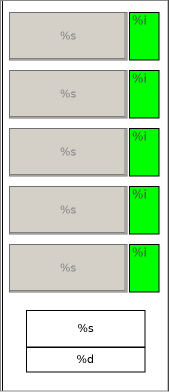
VISUALIZATION VISU_AXE_STD1_FCT_OP  // 169x392
VAR_IN_OUT
	m_Input_MOTEUR: BLOCK_AXE_STD1;
	m_Input_PRG_MOUVEMENT_PS: BLOCK_PRG_MOUVEMENT_PS;
END_VAR
VAR_INPUT
	m_Input_INDEX_MOTEUR : INT;
END_VAR
    RoundedRectangle (2,-1 167x392)
    Rectangle (26,310 119x37), "%s", invisible if: NOT m_Input_PRG_MOUVEMENT_PS.CONF_Balayage[m_Input_INDEX_MOTEUR], text list: 'TextList_Moteurs', text index: 3
    Rectangle (26,347 119x25), "%d", text variable: m_Input_MOTEUR.STATE_NBal, invisible if: NOT m_Input_PRG_MOUVEMENT_PS.CONF_Balayage[m_Input_INDEX_MOTEUR]
    Frame (9,12 152x50)
        shows VISU_FCTS_SA(m_Input_ID_XML := 6, m_Input_Operation := m_Input_MOTEUR.OP_Validation, m_Input_UserRight := PRG_USER.ACTU_USER.FONCTION_SA)
    Frame (9,70 152x50)
        shows VISU_FCTS_SA(m_Input_ID_XML := 7, m_Input_Operation := m_Input_MOTEUR.OP_Stop, m_Input_UserRight := PRG_USER.ACTU_USER.FONCTION_SA)
    Frame (9,128 152x50), invisible if: NOT m_Input_PRG_MOUVEMENT_PS.CONF_Positionnement[m_Input_INDEX_MOTEUR]
        shows VISU_FCTS_SA(m_Input_ID_XML := 8, m_Input_Operation := m_Input_MOTEUR.OP_Position, m_Input_UserRight := PRG_USER.ACTU_USER.FONCTION_SA)
    Frame (9,186 152x50), invisible if: NOT m_Input_PRG_MOUVEMENT_PS.CONF_Rotation[m_Input_INDEX_MOTEUR]
        shows VISU_FCTS_SA(m_Input_ID_XML := 15, m_Input_Operation := m_Input_MOTEUR.OP_Rotation, m_Input_UserRight := PRG_USER.ACTU_USER.FONCTION_SA)
    Frame (9,244 152x50), invisible if: NOT m_Input_PRG_MOUVEMENT_PS.CONF_Balayage[m_Input_INDEX_MOTEUR]
        shows VISU_FCTS_SA(m_Input_ID_XML := 16, m_Input_Operation := m_Input_MOTEUR.OP_Balayage, m_Input_UserRight := PRG_USER.ACTU_USER.FONCTION_SA)
END_VISUALIZATION

// ---- Visualizations/Symbole/MOUVEMENTS PS/AXE STD1/FCT_Part/VISU_AXE_STD1_FCT_OP_OSC.TcVIS
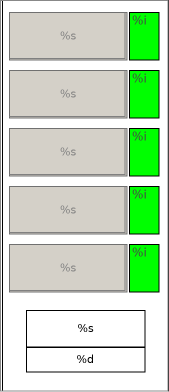
VISUALIZATION VISU_AXE_STD1_FCT_OP_OSC  // 169x392
VAR_IN_OUT
	m_Input_MOTEUR: BLOCK_AXE_STD1_OSCILLANT;
	m_Input_PRG_MOUVEMENT_PS: BLOCK_PRG_MOUVEMENT_PS;
END_VAR
VAR_INPUT
	m_Input_INDEX_MOTEUR : INT;
END_VAR
    RoundedRectangle (2,-1 167x392)
    Rectangle (26,310 119x37), "%s", invisible if: NOT m_Input_PRG_MOUVEMENT_PS.CONF_Balayage[m_Input_INDEX_MOTEUR], text list: 'TextList_Moteurs', text index: 3
    Rectangle (26,347 119x25), "%d", text variable: m_Input_MOTEUR.STATE_NBal, invisible if: NOT m_Input_PRG_MOUVEMENT_PS.CONF_Balayage[m_Input_INDEX_MOTEUR]
    Frame (9,12 152x50)
        shows VISU_FCTS_SA(m_Input_ID_XML := 6, m_Input_Operation := m_Input_MOTEUR.OP_Validation, m_Input_UserRight := PRG_USER.ACTU_USER.FONCTION_SA)
    Frame (9,70 152x50)
        shows VISU_FCTS_SA(m_Input_ID_XML := 7, m_Input_Operation := m_Input_MOTEUR.OP_Stop, m_Input_UserRight := PRG_USER.ACTU_USER.FONCTION_SA)
    Frame (9,128 152x50), invisible if: NOT m_Input_PRG_MOUVEMENT_PS.CONF_Positionnement[m_Input_INDEX_MOTEUR]
        shows VISU_FCTS_SA(m_Input_ID_XML := 8, m_Input_Operation := m_Input_MOTEUR.OP_Position, m_Input_UserRight := PRG_USER.ACTU_USER.FONCTION_SA)
    Frame (9,186 152x50), invisible if: NOT m_Input_PRG_MOUVEMENT_PS.CONF_Rotation[m_Input_INDEX_MOTEUR]
        shows VISU_FCTS_SA(m_Input_ID_XML := 15, m_Input_Operation := m_Input_MOTEUR.OP_Rotation, m_Input_UserRight := PRG_USER.ACTU_USER.FONCTION_SA)
    Frame (9,244 152x50), invisible if: NOT m_Input_PRG_MOUVEMENT_PS.CONF_Balayage[m_Input_INDEX_MOTEUR]
        shows VISU_FCTS_SA(m_Input_ID_XML := 16, m_Input_Operation := m_Input_MOTEUR.OP_Balayage, m_Input_UserRight := PRG_USER.ACTU_USER.FONCTION_SA)
END_VISUALIZATION

// ---- Visualizations/Symbole/MOUVEMENTS PS/AXE STD1/FCT_Part/VISU_AXE_STD1_FCT_TRF.TcVIS
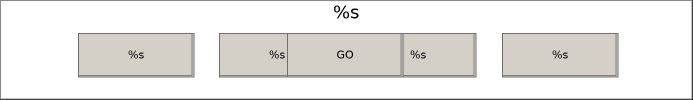
VISUALIZATION VISU_AXE_STD1_FCT_TRF  // 693x100
VAR_IN_OUT
	m_Input_MOTEUR: BLOCK_AXE_STD1;
	m_Input_PRG_MOUVEMENT_PS: BLOCK_PRG_MOUVEMENT_PS;
END_VAR
VAR_INPUT CONSTANT
	m_Input_INDEX_MOTEUR : INT;
	m_Input_Ref_Trf:		USINT;
END_VAR
    Rectangle (0,0 693x100), "%s", text list: 'TextList_Moteurs', text index: 4
    Button (78,33 116x44), "%s", text variable: m_Input_MOTEUR.CONF_ID_Poste[1], invisible if: m_Input_PRG_MOUVEMENT_PS.CONF_NB_POSTE[m_Input_INDEX_MOTEUR]<1, input disabled if: NOT m_Input_MOTEUR.OP_Position.AUTOR_IHM
        OnMouseClick: execute {
            m_Input_MOTEUR.PRM_NPOSTE:=1;
            m_Input_MOTEUR.PRM_NREF:=m_Input_REF_TRF;
            m_Input_MOTEUR.PRM_BalPos:=FALSE;
            m_Input_MOTEUR.PRM_GoToHome:=TRUE;
            m_Input_MOTEUR.PRM_Position:=0;
            m_Input_MOTEUR.OP_POSITION.ON_IHM:=TRUE;
        }
    Button (219,33 116x44), "%s", text variable: m_Input_MOTEUR.CONF_ID_Poste[2], invisible if: m_Input_PRG_MOUVEMENT_PS.CONF_NB_POSTE[m_Input_INDEX_MOTEUR]<2, input disabled if: NOT m_Input_MOTEUR.OP_Position.AUTOR_IHM
        OnMouseClick: execute {
            m_Input_MOTEUR.PRM_NPOSTE:=2;
            m_Input_MOTEUR.PRM_NREF:=m_Input_REF_TRF;
            m_Input_MOTEUR.PRM_BalPos:=FALSE;
            m_Input_MOTEUR.PRM_GoToHome:=TRUE;
            m_Input_MOTEUR.PRM_Position:=0;
            m_Input_MOTEUR.OP_POSITION.ON_IHM:=TRUE;
        }
    Button (360,33 116x44), "%s", text variable: m_Input_MOTEUR.CONF_ID_Poste[3], invisible if: m_Input_PRG_MOUVEMENT_PS.CONF_NB_POSTE[m_Input_INDEX_MOTEUR]<3, input disabled if: NOT m_Input_MOTEUR.OP_Position.AUTOR_IHM
        OnMouseClick: execute {
            m_Input_MOTEUR.PRM_NPOSTE:=3;
            m_Input_MOTEUR.PRM_NREF:=m_Input_REF_TRF;
            m_Input_MOTEUR.PRM_BalPos:=FALSE;
            m_Input_MOTEUR.PRM_GoToHome:=TRUE;
            m_Input_MOTEUR.PRM_Position:=0;
            m_Input_MOTEUR.OP_POSITION.ON_IHM:=TRUE;
        }
    Button (502,33 116x44), "%s", text variable: m_Input_MOTEUR.CONF_ID_Poste[4], invisible if: m_Input_PRG_MOUVEMENT_PS.CONF_NB_POSTE[m_Input_INDEX_MOTEUR]<4, input disabled if: NOT m_Input_MOTEUR.OP_Position.AUTOR_IHM
        OnMouseClick: execute {
            m_Input_MOTEUR.PRM_NPOSTE:=4;
            m_Input_MOTEUR.PRM_NREF:=m_Input_REF_TRF;
            m_Input_MOTEUR.PRM_BalPos:=FALSE;
            m_Input_MOTEUR.PRM_GoToHome:=TRUE;
            m_Input_MOTEUR.PRM_Position:=0;
            m_Input_MOTEUR.OP_POSITION.ON_IHM:=TRUE;
        }
    Button (287,33 116x44), "GO", invisible if: m_Input_PRG_MOUVEMENT_PS.CONF_NB_POSTE[m_Input_INDEX_MOTEUR]<>0, input disabled if: NOT m_Input_MOTEUR.OP_Position.AUTOR_IHM
        OnMouseClick: execute {
            m_Input_MOTEUR.PRM_NPOSTE:=0;
            m_Input_MOTEUR.PRM_NREF:=0;
            m_Input_MOTEUR.PRM_BalPos:=FALSE;
            m_Input_MOTEUR.PRM_GoToHome:=TRUE;
            m_Input_MOTEUR.PRM_Position:=0;
            m_Input_MOTEUR.OP_POSITION.ON_IHM:=TRUE;
        }
END_VISUALIZATION

// ---- Visualizations/Symbole/MOUVEMENTS PS/AXE STD1/FCT_Part/VISU_AXE_STD1_FCT_TRF_OSC.TcVIS
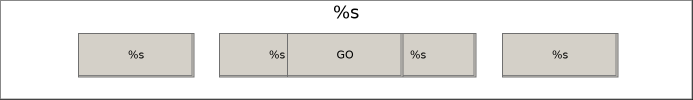
VISUALIZATION VISU_AXE_STD1_FCT_TRF_OSC  // 693x100
VAR_IN_OUT
	m_Input_MOTEUR: BLOCK_AXE_STD1_OSCILLANT;
	m_Input_PRG_MOUVEMENT_PS: BLOCK_PRG_MOUVEMENT_PS;
END_VAR
VAR_INPUT CONSTANT
	m_Input_INDEX_MOTEUR : INT;
	m_Input_Ref_Trf:		USINT;
END_VAR
    Rectangle (0,0 693x100), "%s", text list: 'TextList_Moteurs', text index: 4
    Button (78,33 116x44), "%s", text variable: m_Input_MOTEUR.CONF_ID_Poste[1], invisible if: m_Input_PRG_MOUVEMENT_PS.CONF_NB_POSTE[m_Input_INDEX_MOTEUR]<1, input disabled if: NOT m_Input_MOTEUR.OP_Position.AUTOR_IHM
        OnMouseClick: execute {
            m_Input_MOTEUR.PRM_NPOSTE:=1;
            m_Input_MOTEUR.PRM_NREF:=m_Input_REF_TRF;
            m_Input_MOTEUR.PRM_BalPos:=FALSE;
            m_Input_MOTEUR.PRM_GoToHome:=TRUE;
            m_Input_MOTEUR.PRM_Position:=0;
            m_Input_MOTEUR.OP_POSITION.ON_IHM:=TRUE;
        }
    Button (219,33 116x44), "%s", text variable: m_Input_MOTEUR.CONF_ID_Poste[2], invisible if: m_Input_PRG_MOUVEMENT_PS.CONF_NB_POSTE[m_Input_INDEX_MOTEUR]<2, input disabled if: NOT m_Input_MOTEUR.OP_Position.AUTOR_IHM
        OnMouseClick: execute {
            m_Input_MOTEUR.PRM_NPOSTE:=2;
            m_Input_MOTEUR.PRM_NREF:=m_Input_REF_TRF;
            m_Input_MOTEUR.PRM_BalPos:=FALSE;
            m_Input_MOTEUR.PRM_GoToHome:=TRUE;
            m_Input_MOTEUR.PRM_Position:=0;
            m_Input_MOTEUR.OP_POSITION.ON_IHM:=TRUE;
        }
    Button (360,33 116x44), "%s", text variable: m_Input_MOTEUR.CONF_ID_Poste[3], invisible if: m_Input_PRG_MOUVEMENT_PS.CONF_NB_POSTE[m_Input_INDEX_MOTEUR]<3, input disabled if: NOT m_Input_MOTEUR.OP_Position.AUTOR_IHM
        OnMouseClick: execute {
            m_Input_MOTEUR.PRM_NPOSTE:=3;
            m_Input_MOTEUR.PRM_NREF:=m_Input_REF_TRF;
            m_Input_MOTEUR.PRM_BalPos:=FALSE;
            m_Input_MOTEUR.PRM_GoToHome:=TRUE;
            m_Input_MOTEUR.PRM_Position:=0;
            m_Input_MOTEUR.OP_POSITION.ON_IHM:=TRUE;
        }
    Button (502,33 116x44), "%s", text variable: m_Input_MOTEUR.CONF_ID_Poste[4], invisible if: m_Input_PRG_MOUVEMENT_PS.CONF_NB_POSTE[m_Input_INDEX_MOTEUR]<4, input disabled if: NOT m_Input_MOTEUR.OP_Position.AUTOR_IHM
        OnMouseClick: execute {
            m_Input_MOTEUR.PRM_NPOSTE:=4;
            m_Input_MOTEUR.PRM_NREF:=m_Input_REF_TRF;
            m_Input_MOTEUR.PRM_BalPos:=FALSE;
            m_Input_MOTEUR.PRM_GoToHome:=TRUE;
            m_Input_MOTEUR.PRM_Position:=0;
            m_Input_MOTEUR.OP_POSITION.ON_IHM:=TRUE;
        }
    Button (287,33 116x44), "GO", invisible if: m_Input_PRG_MOUVEMENT_PS.CONF_NB_POSTE[m_Input_INDEX_MOTEUR]<>0, input disabled if: NOT m_Input_MOTEUR.OP_Position.AUTOR_IHM
        OnMouseClick: execute {
            m_Input_MOTEUR.PRM_NPOSTE:=0;
            m_Input_MOTEUR.PRM_NREF:=0;
            m_Input_MOTEUR.PRM_BalPos:=FALSE;
            m_Input_MOTEUR.PRM_GoToHome:=TRUE;
            m_Input_MOTEUR.PRM_Position:=0.0;
            m_Input_MOTEUR.OP_POSITION.ON_IHM:=TRUE;
        }
END_VISUALIZATION

// ---- Visualizations/Symbole/MOUVEMENTS PS/AXE STD1/FCT_Part/VISU_AXE_STD1_LIN_REL_FCT_ETAT.TcVIS
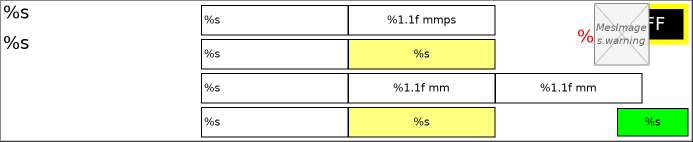
VISUALIZATION VISU_AXE_STD1_LIN_REL_FCT_ETAT  // 693x142
VAR_IN_OUT
	m_Input_MOTEUR: BLOCK_AXE_STD1;
	m_Input_PRG_MOUVEMENT_PS: BLOCK_PRG_MOUVEMENT_PS;
END_VAR
VAR_INPUT
	m_Input_ID_NOM_XML : INT;
END_VAR
    Rectangle (0,0 693x142), "%s", text list: 'TextList_Type_Moteur', text index: m_Input_ID_NOM_XML
    Rectangle (0,28 107x30), "%s", text variable: m_Input_MOTEUR.MNEMO
    RoundedRectangle (201,5 147x30), "%s", text list: 'TextList_Moteurs', text index: 7
    RoundedRectangle (201,39 147x30), "%s", text list: 'TextList_Moteurs', text index: 8
    RoundedRectangle (201,73 147x30), "%s", text list: 'TextList_Moteurs', text index: 9
    RoundedRectangle (201,107 147x30), "%s", text list: 'TextList_Moteurs', text index: 10
    RoundedRectangle (348,5 147x30), "%1.1f mmps", text variable: m_Input_MOTEUR.STATE_Vit
    RoundedRectangle (348,39 147x30), "%s", text variable: m_Input_MOTEUR.CONF_ID_POSTE[m_Input_MOTEUR.PRM_NPOSTE]
    RoundedRectangle (348,73 147x30), "%1.1f mm", text variable: m_Input_MOTEUR.STATE_Pos_Rel
    RoundedRectangle (495,73 147x30), "%1.1f mm", text variable: m_Input_MOTEUR.STATE_Pos
    RoundedRectangle (348,107 147x30), "%s", text variable: m_Input_MOTEUR.CONF_ID_REF[m_Input_MOTEUR.PRM_NRef]
    RoundedRectangle (617,108 71x28), "%s", invisible if: m_Input_MOTEUR.STATE_Homed OR m_Input_MOTEUR.CONF_No_Ref, text list: 'TextList_Moteurs', text index: 11
    RoundedRectangle (617,108 71x28), "%s", invisible if: NOT m_Input_MOTEUR.STATE_Homed OR m_Input_MOTEUR.CONF_No_Ref, text list: 'TextList_Moteurs', text index: 11
    RoundedRectangle (608,4 80x40), invisible if: NOT m_Input_MOTEUR.OP_Validation.OK
    RoundedRectangle (608,4 80x40), invisible if: NOT m_Input_MOTEUR.OP_Validation.AR
    RoundedRectangle (608,4 80x40), invisible if: NOT m_Input_MOTEUR.OP_Validation.EC
    RoundedRectangle (613,9 70x30), "ON", invisible if: m_Input_MOTEUR.STATE_Ar
    RoundedRectangle (613,9 70x30), "OFF", invisible if: NOT m_Input_MOTEUR.STATE_Ar
    Rectangle (535,24 67x21), "%i", text variable: m_Input_MOTEUR.STATE_Err, invisible if: NOT m_Input_MOTEUR.STATE_NOK
    Image (594,3 55x62), invisible if: NOT m_Input_MOTEUR.STATE_NOK, image: MesImages.warning
END_VISUALIZATION

// ---- Visualizations/Symbole/MOUVEMENTS PS/AXE STD1/FCT_Part/VISU_AXE_STD1_LIN_REL_FCT_ETAT_OSC.TcVIS
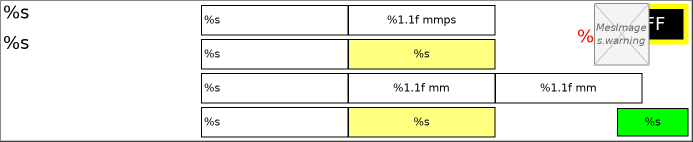
VISUALIZATION VISU_AXE_STD1_LIN_REL_FCT_ETAT_OSC  // 693x142
VAR_IN_OUT
	m_Input_MOTEUR: BLOCK_AXE_STD1_OSCILLANT;
	m_Input_PRG_MOUVEMENT_PS: BLOCK_PRG_MOUVEMENT_PS;
END_VAR
VAR_INPUT
	m_Input_ID_NOM_XML : INT;
END_VAR
    Rectangle (0,0 693x142), "%s", text list: 'TextList_Type_Moteur', text index: m_Input_ID_NOM_XML
    Rectangle (0,28 107x30), "%s", text variable: m_Input_MOTEUR.MNEMO
    RoundedRectangle (201,5 147x30), "%s", text list: 'TextList_Moteurs', text index: 7
    RoundedRectangle (201,39 147x30), "%s", text list: 'TextList_Moteurs', text index: 8
    RoundedRectangle (201,73 147x30), "%s", text list: 'TextList_Moteurs', text index: 9
    RoundedRectangle (201,107 147x30), "%s", text list: 'TextList_Moteurs', text index: 10
    RoundedRectangle (348,5 147x30), "%1.1f mmps", text variable: m_Input_MOTEUR.STATE_Vit
    RoundedRectangle (348,39 147x30), "%s", text variable: m_Input_MOTEUR.CONF_ID_POSTE[m_Input_MOTEUR.PRM_NPOSTE]
    RoundedRectangle (348,73 147x30), "%1.1f mm", text variable: m_Input_MOTEUR.STATE_Pos_Rel
    RoundedRectangle (495,73 147x30), "%1.1f mm", text variable: m_Input_MOTEUR.STATE_Pos
    RoundedRectangle (348,107 147x30), "%s", text variable: m_Input_MOTEUR.CONF_ID_REF[m_Input_MOTEUR.PRM_NRef]
    RoundedRectangle (617,108 71x28), "%s", invisible if: m_Input_MOTEUR.STATE_Homed OR m_Input_MOTEUR.CONF_No_Ref, text list: 'TextList_Moteurs', text index: 11
    RoundedRectangle (617,108 71x28), "%s", invisible if: NOT m_Input_MOTEUR.STATE_Homed OR m_Input_MOTEUR.CONF_No_Ref, text list: 'TextList_Moteurs', text index: 11
    RoundedRectangle (608,4 80x40), invisible if: NOT m_Input_MOTEUR.OP_Validation.OK
    RoundedRectangle (608,4 80x40), invisible if: NOT m_Input_MOTEUR.OP_Validation.AR
    RoundedRectangle (608,4 80x40), invisible if: NOT m_Input_MOTEUR.OP_Validation.EC
    RoundedRectangle (613,9 70x30), "ON", invisible if: m_Input_MOTEUR.STATE_Ar
    RoundedRectangle (613,9 70x30), "OFF", invisible if: NOT m_Input_MOTEUR.STATE_Ar
    Rectangle (535,24 67x21), "%i", text variable: m_Input_MOTEUR.STATE_Err, invisible if: NOT m_Input_MOTEUR.STATE_NOK
    Image (594,3 55x62), invisible if: NOT m_Input_MOTEUR.STATE_NOK, image: MesImages.warning
END_VISUALIZATION

// ---- Visualizations/Symbole/MOUVEMENTS PS/AXE STD1/FCT_Part/VISU_AXE_STD1_LIN_ROT_FCT_CONS.TcVIS
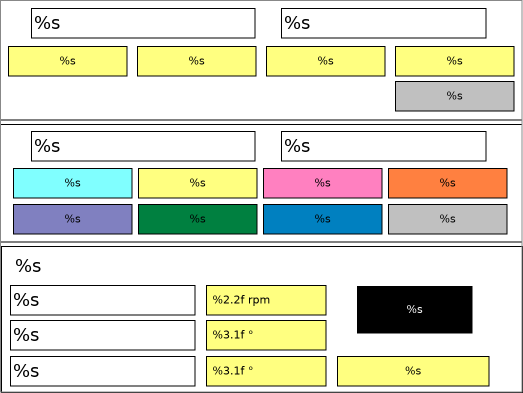
VISUALIZATION VISU_AXE_STD1_LIN_ROT_FCT_CONS  // 523x393
VAR_IN_OUT
	m_Input_MOTEUR: BLOCK_AXE_STD1;
	m_Input_PRG_MOUVEMENT_PS: BLOCK_PRG_MOUVEMENT_PS;
END_VAR
VAR_INPUT CONSTANT
	m_Input_INDEX_MOTEUR : INT;
END_VAR
    Rectangle (0,0 522x120)
    RoundedRectangle (31,8 224x30), "%s", text list: 'TextList_Moteurs', text index: 13
    RoundedRectangle (281,8 205x30), "%s", text variable: m_Input_MOTEUR.CONF_ID_Poste[m_Input_MOTEUR.PRM_NPoste]
    RoundedRectangle (8,46 119x30), "%s", text variable: m_Input_MOTEUR.CONF_ID_Poste[1], invisible if: m_Input_PRG_MOUVEMENT_PS.CONF_NB_POSTE[m_Input_INDEX_MOTEUR]<1, input disabled if: (NOT PRG_User.ACTU_USER.MAINTENANCE AND m_Input_MOTEUR.MANUAL) OR (NOT PRG_User.ACTU_USER.FONCTION_SA AND NOT m_Input_MOTEUR.MANUAL)
        OnMouseClick: execute { m_Input_MOTEUR.PRM_NPOSTE:=1; }
    RoundedRectangle (395,81 119x30), "%s", text variable: m_Input_MOTEUR.CONF_ID_POSTE[0], invisible if: NOT m_Input_PRG_MOUVEMENT_PS.CONF_Use_Poste0[m_Input_INDEX_MOTEUR], input disabled if: (NOT PRG_User.ACTU_USER.MAINTENANCE AND m_Input_MOTEUR.MANUAL) OR (NOT PRG_User.ACTU_USER.FONCTION_SA AND NOT m_Input_MOTEUR.MANUAL)
        OnMouseClick: execute { m_Input_MOTEUR.PRM_NPOSTE:=0; }
    RoundedRectangle (137,46 119x30), "%s", text variable: m_Input_MOTEUR.CONF_ID_Poste[2], invisible if: m_Input_PRG_MOUVEMENT_PS.CONF_NB_POSTE[m_Input_INDEX_MOTEUR]<2, input disabled if: (NOT PRG_User.ACTU_USER.MAINTENANCE AND m_Input_MOTEUR.MANUAL) OR (NOT PRG_User.ACTU_USER.FONCTION_SA AND NOT m_Input_MOTEUR.MANUAL)
        OnMouseClick: execute { m_Input_MOTEUR.PRM_NPOSTE:=2; }
    RoundedRectangle (266,46 119x30), "%s", text variable: m_Input_MOTEUR.CONF_ID_Poste[3], invisible if: m_Input_PRG_MOUVEMENT_PS.CONF_NB_POSTE[m_Input_INDEX_MOTEUR]<3, input disabled if: (NOT PRG_User.ACTU_USER.MAINTENANCE AND m_Input_MOTEUR.MANUAL) OR (NOT PRG_User.ACTU_USER.FONCTION_SA AND NOT m_Input_MOTEUR.MANUAL)
        OnMouseClick: execute { m_Input_MOTEUR.PRM_NPOSTE:=3; }
    RoundedRectangle (395,46 119x30), "%s", text variable: m_Input_MOTEUR.CONF_ID_Poste[4], invisible if: m_Input_PRG_MOUVEMENT_PS.CONF_NB_POSTE[m_Input_INDEX_MOTEUR]<4, input disabled if: (NOT PRG_User.ACTU_USER.MAINTENANCE AND m_Input_MOTEUR.MANUAL) OR (NOT PRG_User.ACTU_USER.FONCTION_SA AND NOT m_Input_MOTEUR.MANUAL)
        OnMouseClick: execute { m_Input_MOTEUR.PRM_NPOSTE:=4; }
    Rectangle (0,124 522x118)
    RoundedRectangle (31,131 224x30), "%s", text list: 'TextList_Moteurs', text index: 14
    RoundedRectangle (281,131 205x30), "%s", text variable: m_Input_MOTEUR.CONF_ID_Ref[m_Input_MOTEUR.PRM_NRef]
    RoundedRectangle (13,168 119x30), "%s", text variable: m_Input_MOTEUR.CONF_ID_REF[1], invisible if: m_Input_PRG_MOUVEMENT_PS.CONF_NB_REF[m_Input_INDEX_MOTEUR]<1, input disabled if: (NOT PRG_User.ACTU_USER.MAINTENANCE AND m_Input_MOTEUR.MANUAL) OR (NOT PRG_User.ACTU_USER.FONCTION_SA AND NOT m_Input_MOTEUR.MANUAL)
        OnMouseClick: execute { m_Input_MOTEUR.PRM_NREF:=1; }
    RoundedRectangle (138,168 119x30), "%s", text variable: m_Input_MOTEUR.CONF_ID_REF[2], invisible if: m_Input_PRG_MOUVEMENT_PS.CONF_NB_REF[m_Input_INDEX_MOTEUR]<2, input disabled if: (NOT PRG_User.ACTU_USER.MAINTENANCE AND m_Input_MOTEUR.MANUAL) OR (NOT PRG_User.ACTU_USER.FONCTION_SA AND NOT m_Input_MOTEUR.MANUAL)
        OnMouseClick: execute { m_Input_MOTEUR.PRM_NREF:=2; }
    RoundedRectangle (263,168 119x30), "%s", text variable: m_Input_MOTEUR.CONF_ID_REF[3], invisible if: m_Input_PRG_MOUVEMENT_PS.CONF_NB_REF[m_Input_INDEX_MOTEUR]<3, input disabled if: (NOT PRG_User.ACTU_USER.MAINTENANCE AND m_Input_MOTEUR.MANUAL) OR (NOT PRG_User.ACTU_USER.FONCTION_SA AND NOT m_Input_MOTEUR.MANUAL)
        OnMouseUp: execute { m_Input_MOTEUR.PRM_NREF:=3; }
    RoundedRectangle (388,168 119x30), "%s", text variable: m_Input_MOTEUR.CONF_ID_REF[4], invisible if: m_Input_PRG_MOUVEMENT_PS.CONF_NB_REF[m_Input_INDEX_MOTEUR]<4, input disabled if: (NOT PRG_User.ACTU_USER.MAINTENANCE AND m_Input_MOTEUR.MANUAL) OR (NOT PRG_User.ACTU_USER.FONCTION_SA AND NOT m_Input_MOTEUR.MANUAL)
        OnMouseClick: execute { m_Input_MOTEUR.PRM_NREF:=4; }
    RoundedRectangle (13,204 119x30), "%s", text variable: m_Input_MOTEUR.CONF_ID_REF[5], invisible if: m_Input_PRG_MOUVEMENT_PS.CONF_NB_REF[m_Input_INDEX_MOTEUR]<5, input disabled if: (NOT PRG_User.ACTU_USER.MAINTENANCE AND m_Input_MOTEUR.MANUAL) OR (NOT PRG_User.ACTU_USER.FONCTION_SA AND NOT m_Input_MOTEUR.MANUAL)
        OnMouseClick: execute { m_Input_MOTEUR.PRM_NREF:=5; }
    RoundedRectangle (138,204 119x30), "%s", text variable: m_Input_MOTEUR.CONF_ID_REF[6], invisible if: m_Input_PRG_MOUVEMENT_PS.CONF_NB_REF[m_Input_INDEX_MOTEUR]<6, input disabled if: (NOT PRG_User.ACTU_USER.MAINTENANCE AND m_Input_MOTEUR.MANUAL) OR (NOT PRG_User.ACTU_USER.FONCTION_SA AND NOT m_Input_MOTEUR.MANUAL)
        OnMouseClick: execute { m_Input_MOTEUR.PRM_NREF:=6; }
    RoundedRectangle (388,204 119x30), "%s", text variable: m_Input_MOTEUR.CONF_ID_REF[0], invisible if: NOT m_Input_PRG_MOUVEMENT_PS.CONF_Use_Ref0[m_Input_INDEX_MOTEUR], input disabled if: (NOT PRG_User.ACTU_USER.MAINTENANCE AND m_Input_MOTEUR.MANUAL) OR (NOT PRG_User.ACTU_USER.FONCTION_SA AND NOT m_Input_MOTEUR.MANUAL)
        OnMouseClick: execute { m_Input_MOTEUR.PRM_NREF:=0; }
    RoundedRectangle (263,204 119x30), "%s", text variable: m_Input_MOTEUR.CONF_ID_REF[7], invisible if: m_Input_PRG_MOUVEMENT_PS.CONF_NB_REF[m_Input_INDEX_MOTEUR]<7, input disabled if: (NOT PRG_User.ACTU_USER.MAINTENANCE AND m_Input_MOTEUR.MANUAL) OR (NOT PRG_User.ACTU_USER.FONCTION_SA AND NOT m_Input_MOTEUR.MANUAL)
        OnMouseClick: execute { m_Input_MOTEUR.PRM_NREF:=7; }
    Rectangle (1,246 522x147)
    RoundedRectangle (10,320 185x30), "%s", invisible if: NOT m_Input_PRG_MOUVEMENT_PS.CONF_Balayage[m_Input_INDEX_MOTEUR] AND NOT m_Input_PRG_MOUVEMENT_PS.CONF_Positionnement[m_Input_INDEX_MOTEUR], text list: 'TextList_Moteurs', text index: 12
    RoundedRectangle (206,320 120x30), "%3.1f mm", text variable: m_Input_MOTEUR.PRM_Position, invisible if: (NOT m_Input_PRG_MOUVEMENT_PS.CONF_Balayage[m_Input_INDEX_MOTEUR] AND NOT m_Input_PRG_MOUVEMENT_PS.CONF_Positionnement[m_Input_INDEX_MOTEUR]) OR NOT m_Input_MOTEUR.CONF_Mvt_Lineaire, input disabled if: (NOT PRG_User.ACTU_USER.MAINTENANCE AND m_Input_MOTEUR.MANUAL) OR (NOT PRG_User.ACTU_USER.FONCTION_SA AND NOT m_Input_MOTEUR.MANUAL)
        OnMouseClick: write the text variable via VisuDialogs.Numpad, min m_Input_PRG_MOUVEMENT_PS.CONF_MIN_POS[m_Input_INDEX_MOTEUR], max m_Input_PRG_MOUVEMENT_PS.CONF_MAX_POS[m_Input_INDEX_MOTEUR]
    RoundedRectangle (10,285 185x30), "%s", invisible if: NOT m_Input_PRG_MOUVEMENT_PS.CONF_Balayage[m_Input_INDEX_MOTEUR] AND NOT m_Input_PRG_MOUVEMENT_PS.CONF_Rotation[m_Input_INDEX_MOTEUR], text list: 'TextList_Moteurs', text index: 7
    RoundedRectangle (206,285 120x30), "%2.2f mmps", text variable: m_Input_MOTEUR.PRM_V_BalRot, invisible if: (NOT m_Input_PRG_MOUVEMENT_PS.CONF_Balayage[m_Input_INDEX_MOTEUR] AND NOT m_Input_PRG_MOUVEMENT_PS.CONF_Rotation[m_Input_INDEX_MOTEUR]) OR NOT m_Input_MOTEUR.CONF_Mvt_Lineaire, input disabled if: (NOT PRG_User.ACTU_USER.MAINTENANCE AND m_Input_MOTEUR.MANUAL) OR (NOT PRG_User.ACTU_USER.FONCTION_SA AND NOT m_Input_MOTEUR.MANUAL)
        OnMouseClick: write the text variable via VisuDialogs.Numpad, min m_Input_PRG_MOUVEMENT_PS.CONF_MIN_SPEED[m_Input_INDEX_MOTEUR], max m_Input_PRG_MOUVEMENT_PS.CONF_MAX_SPEED[m_Input_INDEX_MOTEUR]
    RoundedRectangle (10,356 185x30), "%s", invisible if: NOT m_Input_PRG_MOUVEMENT_PS.CONF_Balayage[m_Input_INDEX_MOTEUR], text list: 'TextList_Moteurs', text index: 16
    RoundedRectangle (206,356 120x30), "%3.1f mm", text variable: m_Input_MOTEUR.PRM_Angle_Bal, invisible if: NOT m_Input_PRG_MOUVEMENT_PS.CONF_Balayage[m_Input_INDEX_MOTEUR] OR NOT m_Input_MOTEUR.CONF_Mvt_Lineaire, input disabled if: (NOT PRG_User.ACTU_USER.MAINTENANCE AND m_Input_MOTEUR.MANUAL) OR (NOT PRG_User.ACTU_USER.FONCTION_SA AND NOT m_Input_MOTEUR.MANUAL)
        OnMouseClick: write the text variable via VisuDialogs.Numpad
    RoundedRectangle (357,286 115x47), "%s", invisible if: NOT m_Input_MOTEUR.PRM_GotoHome OR NOT m_Input_PRG_MOUVEMENT_PS.CONF_POSITIONNEMENT[m_Input_INDEX_MOTEUR], input disabled if: (NOT PRG_User.ACTU_USER.MAINTENANCE AND m_Input_MOTEUR.MANUAL) OR (NOT PRG_User.ACTU_USER.FONCTION_SA AND NOT m_Input_MOTEUR.MANUAL), text list: 'TextList_Moteurs', text index: 19
        toggle m_Input_MOTEUR.PRM_GoToHome
    RoundedRectangle (357,286 115x47), "%s", invisible if: m_Input_MOTEUR.PRM_Gotohome OR NOT m_Input_PRG_MOUVEMENT_PS.CONF_POSITIONNEMENT[m_Input_INDEX_MOTEUR], input disabled if: (NOT PRG_User.ACTU_USER.MAINTENANCE AND m_Input_MOTEUR.MANUAL) OR (NOT PRG_User.ACTU_USER.FONCTION_SA AND NOT m_Input_MOTEUR.MANUAL), text list: 'TextList_Moteurs', text index: 20
        toggle m_Input_MOTEUR.PRM_GoToHome
    RoundedRectangle (337,356 152x30), "%s", invisible if: NOT m_Input_PRG_MOUVEMENT_PS.CONF_Balayage[m_Input_INDEX_MOTEUR] OR NOT m_Input_MOTEUR.PRM_BalPos, input disabled if: (NOT PRG_User.ACTU_USER.MAINTENANCE AND m_Input_MOTEUR.MANUAL) OR (NOT PRG_User.ACTU_USER.FONCTION_SA AND NOT m_Input_MOTEUR.MANUAL), text list: 'TextList_Moteurs', text index: 21
        toggle m_Input_MOTEUR.PRM_BalPos
    RoundedRectangle (337,356 152x30), "%s", invisible if: NOT m_Input_PRG_MOUVEMENT_PS.CONF_Balayage[m_Input_INDEX_MOTEUR] OR m_Input_MOTEUR.PRM_BalPos, input disabled if: (NOT PRG_User.ACTU_USER.MAINTENANCE AND m_Input_MOTEUR.MANUAL) OR (NOT PRG_User.ACTU_USER.FONCTION_SA AND NOT m_Input_MOTEUR.MANUAL), text list: 'TextList_Process', text index: 22
        toggle m_Input_MOTEUR.PRM_BalPos
    RoundedRectangle (12,251 390x30), "%s", text list: 'TextList_Moteurs', text index: 15
    RoundedRectangle (206,285 120x30), "%2.2f rpm", text variable: m_Input_MOTEUR.PRM_V_BalRot, invisible if: (NOT m_Input_PRG_MOUVEMENT_PS.CONF_Balayage[m_Input_INDEX_MOTEUR] AND NOT m_Input_PRG_MOUVEMENT_PS.CONF_Rotation[m_Input_INDEX_MOTEUR]) OR m_Input_MOTEUR.CONF_Mvt_Lineaire, input disabled if: (NOT PRG_User.ACTU_USER.MAINTENANCE AND m_Input_MOTEUR.MANUAL) OR (NOT PRG_User.ACTU_USER.FONCTION_SA AND NOT m_Input_MOTEUR.MANUAL)
        OnMouseClick: write the text variable via VisuDialogs.Numpad, min m_Input_PRG_MOUVEMENT_PS.CONF_MIN_SPEED[m_Input_INDEX_MOTEUR], max m_Input_PRG_MOUVEMENT_PS.CONF_MAX_SPEED[m_Input_INDEX_MOTEUR]
    RoundedRectangle (206,320 120x30), "%3.1f °", text variable: m_Input_MOTEUR.PRM_Position, invisible if: (NOT m_Input_PRG_MOUVEMENT_PS.CONF_Balayage[m_Input_INDEX_MOTEUR] AND NOT m_Input_PRG_MOUVEMENT_PS.CONF_Positionnement[m_Input_INDEX_MOTEUR]) OR m_Input_MOTEUR.CONF_Mvt_Lineaire, input disabled if: (NOT PRG_User.ACTU_USER.MAINTENANCE AND m_Input_MOTEUR.MANUAL) OR (NOT PRG_User.ACTU_USER.FONCTION_SA AND NOT m_Input_MOTEUR.MANUAL)
        OnMouseClick: write the text variable via VisuDialogs.Numpad, min m_Input_PRG_MOUVEMENT_PS.CONF_MIN_POS[m_Input_INDEX_MOTEUR], max m_Input_PRG_MOUVEMENT_PS.CONF_MAX_POS[m_Input_INDEX_MOTEUR]
    RoundedRectangle (206,356 120x30), "%3.1f °", text variable: m_Input_MOTEUR.PRM_Angle_Bal, invisible if: NOT m_Input_PRG_MOUVEMENT_PS.CONF_Balayage[m_Input_INDEX_MOTEUR] OR m_Input_MOTEUR.CONF_Mvt_Lineaire, input disabled if: (NOT PRG_User.ACTU_USER.MAINTENANCE AND m_Input_MOTEUR.MANUAL) OR (NOT PRG_User.ACTU_USER.FONCTION_SA AND NOT m_Input_MOTEUR.MANUAL)
        OnMouseClick: write the text variable via VisuDialogs.Numpad, min 0, max 360
END_VISUALIZATION

// ---- Visualizations/Symbole/MOUVEMENTS PS/AXE STD1/FCT_Part/VISU_AXE_STD1_LIN_ROT_FCT_CONS_OSC.TcVIS
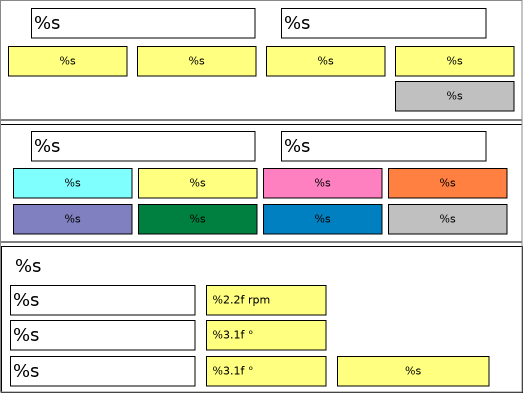
VISUALIZATION VISU_AXE_STD1_LIN_ROT_FCT_CONS_OSC  // 523x393
VAR_IN_OUT
	m_Input_MOTEUR: BLOCK_AXE_STD1_OSCILLANT;
	m_Input_PRG_MOUVEMENT_PS: BLOCK_PRG_MOUVEMENT_PS;
END_VAR
VAR_INPUT CONSTANT
	m_Input_INDEX_MOTEUR : INT;
END_VAR
    Rectangle (0,0 522x120)
    RoundedRectangle (31,8 224x30), "%s", text list: 'TextList_Moteurs', text index: 13
    RoundedRectangle (281,8 205x30), "%s", text variable: m_Input_MOTEUR.CONF_ID_Poste[m_Input_MOTEUR.PRM_NPoste]
    RoundedRectangle (8,46 119x30), "%s", text variable: m_Input_MOTEUR.CONF_ID_Poste[1], invisible if: m_Input_PRG_MOUVEMENT_PS.CONF_NB_POSTE[m_Input_INDEX_MOTEUR]<1, input disabled if: (NOT PRG_User.ACTU_USER.MAINTENANCE AND m_Input_MOTEUR.MANUAL) OR (NOT PRG_User.ACTU_USER.FONCTION_SA AND NOT m_Input_MOTEUR.MANUAL)
        OnMouseClick: execute { m_Input_MOTEUR.PRM_NPOSTE:=1; }
    RoundedRectangle (395,81 119x30), "%s", text variable: m_Input_MOTEUR.CONF_ID_POSTE[0], invisible if: NOT m_Input_PRG_MOUVEMENT_PS.CONF_Use_Poste0[m_Input_INDEX_MOTEUR], input disabled if: (NOT PRG_User.ACTU_USER.MAINTENANCE AND m_Input_MOTEUR.MANUAL) OR (NOT PRG_User.ACTU_USER.FONCTION_SA AND NOT m_Input_MOTEUR.MANUAL)
        OnMouseClick: execute { m_Input_MOTEUR.PRM_NPOSTE:=0; }
    RoundedRectangle (137,46 119x30), "%s", text variable: m_Input_MOTEUR.CONF_ID_Poste[2], invisible if: m_Input_PRG_MOUVEMENT_PS.CONF_NB_POSTE[m_Input_INDEX_MOTEUR]<2, input disabled if: (NOT PRG_User.ACTU_USER.MAINTENANCE AND m_Input_MOTEUR.MANUAL) OR (NOT PRG_User.ACTU_USER.FONCTION_SA AND NOT m_Input_MOTEUR.MANUAL)
        OnMouseClick: execute { m_Input_MOTEUR.PRM_NPOSTE:=2; }
    RoundedRectangle (266,46 119x30), "%s", text variable: m_Input_MOTEUR.CONF_ID_Poste[3], invisible if: m_Input_PRG_MOUVEMENT_PS.CONF_NB_POSTE[m_Input_INDEX_MOTEUR]<3, input disabled if: (NOT PRG_User.ACTU_USER.MAINTENANCE AND m_Input_MOTEUR.MANUAL) OR (NOT PRG_User.ACTU_USER.FONCTION_SA AND NOT m_Input_MOTEUR.MANUAL)
        OnMouseClick: execute { m_Input_MOTEUR.PRM_NPOSTE:=3; }
    RoundedRectangle (395,46 119x30), "%s", text variable: m_Input_MOTEUR.CONF_ID_Poste[4], invisible if: m_Input_PRG_MOUVEMENT_PS.CONF_NB_POSTE[m_Input_INDEX_MOTEUR]<4, input disabled if: (NOT PRG_User.ACTU_USER.MAINTENANCE AND m_Input_MOTEUR.MANUAL) OR (NOT PRG_User.ACTU_USER.FONCTION_SA AND NOT m_Input_MOTEUR.MANUAL)
        OnMouseClick: execute { m_Input_MOTEUR.PRM_NPOSTE:=4; }
    Rectangle (0,124 522x118)
    RoundedRectangle (31,131 224x30), "%s", text list: 'TextList_Moteurs', text index: 14
    RoundedRectangle (281,131 205x30), "%s", text variable: m_Input_MOTEUR.CONF_ID_Ref[m_Input_MOTEUR.PRM_NRef]
    RoundedRectangle (13,168 119x30), "%s", text variable: m_Input_MOTEUR.CONF_ID_REF[1], invisible if: m_Input_PRG_MOUVEMENT_PS.CONF_NB_REF[m_Input_INDEX_MOTEUR]<1, input disabled if: (NOT PRG_User.ACTU_USER.MAINTENANCE AND m_Input_MOTEUR.MANUAL) OR (NOT PRG_User.ACTU_USER.FONCTION_SA AND NOT m_Input_MOTEUR.MANUAL)
        OnMouseClick: execute { m_Input_MOTEUR.PRM_NREF:=1; }
    RoundedRectangle (138,168 119x30), "%s", text variable: m_Input_MOTEUR.CONF_ID_REF[2], invisible if: m_Input_PRG_MOUVEMENT_PS.CONF_NB_REF[m_Input_INDEX_MOTEUR]<2, input disabled if: (NOT PRG_User.ACTU_USER.MAINTENANCE AND m_Input_MOTEUR.MANUAL) OR (NOT PRG_User.ACTU_USER.FONCTION_SA AND NOT m_Input_MOTEUR.MANUAL)
        OnMouseClick: execute { m_Input_MOTEUR.PRM_NREF:=2; }
    RoundedRectangle (263,168 119x30), "%s", text variable: m_Input_MOTEUR.CONF_ID_REF[3], invisible if: m_Input_PRG_MOUVEMENT_PS.CONF_NB_REF[m_Input_INDEX_MOTEUR]<3, input disabled if: (NOT PRG_User.ACTU_USER.MAINTENANCE AND m_Input_MOTEUR.MANUAL) OR (NOT PRG_User.ACTU_USER.FONCTION_SA AND NOT m_Input_MOTEUR.MANUAL)
        OnMouseUp: execute { m_Input_MOTEUR.PRM_NREF:=3; }
    RoundedRectangle (388,168 119x30), "%s", text variable: m_Input_MOTEUR.CONF_ID_REF[4], invisible if: m_Input_PRG_MOUVEMENT_PS.CONF_NB_REF[m_Input_INDEX_MOTEUR]<4, input disabled if: (NOT PRG_User.ACTU_USER.MAINTENANCE AND m_Input_MOTEUR.MANUAL) OR (NOT PRG_User.ACTU_USER.FONCTION_SA AND NOT m_Input_MOTEUR.MANUAL)
        OnMouseClick: execute { m_Input_MOTEUR.PRM_NREF:=4; }
    RoundedRectangle (13,204 119x30), "%s", text variable: m_Input_MOTEUR.CONF_ID_REF[5], invisible if: m_Input_PRG_MOUVEMENT_PS.CONF_NB_REF[m_Input_INDEX_MOTEUR]<5, input disabled if: (NOT PRG_User.ACTU_USER.MAINTENANCE AND m_Input_MOTEUR.MANUAL) OR (NOT PRG_User.ACTU_USER.FONCTION_SA AND NOT m_Input_MOTEUR.MANUAL)
        OnMouseClick: execute { m_Input_MOTEUR.PRM_NREF:=5; }
    RoundedRectangle (138,204 119x30), "%s", text variable: m_Input_MOTEUR.CONF_ID_REF[6], invisible if: m_Input_PRG_MOUVEMENT_PS.CONF_NB_REF[m_Input_INDEX_MOTEUR]<6, input disabled if: (NOT PRG_User.ACTU_USER.MAINTENANCE AND m_Input_MOTEUR.MANUAL) OR (NOT PRG_User.ACTU_USER.FONCTION_SA AND NOT m_Input_MOTEUR.MANUAL)
        OnMouseClick: execute { m_Input_MOTEUR.PRM_NREF:=6; }
    RoundedRectangle (388,204 119x30), "%s", text variable: m_Input_MOTEUR.CONF_ID_REF[0], invisible if: NOT m_Input_PRG_MOUVEMENT_PS.CONF_Use_Ref0[m_Input_INDEX_MOTEUR], input disabled if: (NOT PRG_User.ACTU_USER.MAINTENANCE AND m_Input_MOTEUR.MANUAL) OR (NOT PRG_User.ACTU_USER.FONCTION_SA AND NOT m_Input_MOTEUR.MANUAL)
        OnMouseClick: execute { m_Input_MOTEUR.PRM_NREF:=0; }
    RoundedRectangle (263,204 119x30), "%s", text variable: m_Input_MOTEUR.CONF_ID_REF[7], invisible if: m_Input_PRG_MOUVEMENT_PS.CONF_NB_REF[m_Input_INDEX_MOTEUR]<7, input disabled if: (NOT PRG_User.ACTU_USER.MAINTENANCE AND m_Input_MOTEUR.MANUAL) OR (NOT PRG_User.ACTU_USER.FONCTION_SA AND NOT m_Input_MOTEUR.MANUAL)
        OnMouseClick: execute { m_Input_MOTEUR.PRM_NREF:=7; }
    Rectangle (1,246 522x147)
    RoundedRectangle (10,320 185x30), "%s", invisible if: NOT m_Input_PRG_MOUVEMENT_PS.CONF_Balayage[m_Input_INDEX_MOTEUR] AND NOT m_Input_PRG_MOUVEMENT_PS.CONF_Positionnement[m_Input_INDEX_MOTEUR], text list: 'TextList_Moteurs', text index: 12
    RoundedRectangle (206,320 120x30), "%3.1f mm", text variable: m_Input_MOTEUR.PRM_Position, invisible if: (NOT m_Input_PRG_MOUVEMENT_PS.CONF_Balayage[m_Input_INDEX_MOTEUR] AND NOT m_Input_PRG_MOUVEMENT_PS.CONF_Positionnement[m_Input_INDEX_MOTEUR]) OR NOT m_Input_MOTEUR.CONF_Mvt_Lineaire, input disabled if: (NOT PRG_User.ACTU_USER.MAINTENANCE AND m_Input_MOTEUR.MANUAL) OR (NOT PRG_User.ACTU_USER.FONCTION_SA AND NOT m_Input_MOTEUR.MANUAL)
        OnMouseClick: write the text variable via VisuDialogs.Numpad, min m_Input_PRG_MOUVEMENT_PS.CONF_MIN_POS[m_Input_INDEX_MOTEUR], max m_Input_PRG_MOUVEMENT_PS.CONF_MAX_POS[m_Input_INDEX_MOTEUR]
    RoundedRectangle (10,285 185x30), "%s", invisible if: NOT m_Input_PRG_MOUVEMENT_PS.CONF_Balayage[m_Input_INDEX_MOTEUR] AND NOT m_Input_PRG_MOUVEMENT_PS.CONF_Rotation[m_Input_INDEX_MOTEUR], text list: 'TextList_Moteurs', text index: 7
    RoundedRectangle (206,285 120x30), "%2.2f mmps", text variable: m_Input_MOTEUR.PRM_V_BalRot, invisible if: (NOT m_Input_PRG_MOUVEMENT_PS.CONF_Balayage[m_Input_INDEX_MOTEUR] AND NOT m_Input_PRG_MOUVEMENT_PS.CONF_Rotation[m_Input_INDEX_MOTEUR]) OR NOT m_Input_MOTEUR.CONF_Mvt_Lineaire, input disabled if: (NOT PRG_User.ACTU_USER.MAINTENANCE AND m_Input_MOTEUR.MANUAL) OR (NOT PRG_User.ACTU_USER.FONCTION_SA AND NOT m_Input_MOTEUR.MANUAL)
        OnMouseClick: write the text variable via VisuDialogs.Numpad, min m_Input_PRG_MOUVEMENT_PS.CONF_MIN_SPEED[m_Input_INDEX_MOTEUR], max m_Input_PRG_MOUVEMENT_PS.CONF_MAX_SPEED[m_Input_INDEX_MOTEUR]
    RoundedRectangle (10,356 185x30), "%s", invisible if: NOT m_Input_PRG_MOUVEMENT_PS.CONF_Balayage[m_Input_INDEX_MOTEUR], text list: 'TextList_Moteurs', text index: 16
    RoundedRectangle (206,356 120x30), "%3.1f mm", text variable: m_Input_MOTEUR.PRM_Angle_Bal, invisible if: NOT m_Input_PRG_MOUVEMENT_PS.CONF_Balayage[m_Input_INDEX_MOTEUR] OR NOT m_Input_MOTEUR.CONF_Mvt_Lineaire, input disabled if: (NOT PRG_User.ACTU_USER.MAINTENANCE AND m_Input_MOTEUR.MANUAL) OR (NOT PRG_User.ACTU_USER.FONCTION_SA AND NOT m_Input_MOTEUR.MANUAL)
        OnMouseClick: write the text variable via VisuDialogs.Numpad
    RoundedRectangle (337,356 152x30), "%s", invisible if: NOT m_Input_PRG_MOUVEMENT_PS.CONF_Balayage[m_Input_INDEX_MOTEUR] OR NOT m_Input_MOTEUR.PRM_BalPos, input disabled if: (NOT PRG_User.ACTU_USER.MAINTENANCE AND m_Input_MOTEUR.MANUAL) OR (NOT PRG_User.ACTU_USER.FONCTION_SA AND NOT m_Input_MOTEUR.MANUAL), text list: 'TextList_Moteurs', text index: 21
        toggle m_Input_MOTEUR.PRM_BalPos
    RoundedRectangle (337,356 152x30), "%s", invisible if: NOT m_Input_PRG_MOUVEMENT_PS.CONF_Balayage[m_Input_INDEX_MOTEUR] OR m_Input_MOTEUR.PRM_BalPos, input disabled if: (NOT PRG_User.ACTU_USER.MAINTENANCE AND m_Input_MOTEUR.MANUAL) OR (NOT PRG_User.ACTU_USER.FONCTION_SA AND NOT m_Input_MOTEUR.MANUAL), text list: 'TextList_Process', text index: 22
        toggle m_Input_MOTEUR.PRM_BalPos
    RoundedRectangle (12,251 390x30), "%s", text list: 'TextList_Moteurs', text index: 15
    RoundedRectangle (206,285 120x30), "%2.2f rpm", text variable: m_Input_MOTEUR.PRM_V_BalRot, invisible if: (NOT m_Input_PRG_MOUVEMENT_PS.CONF_Balayage[m_Input_INDEX_MOTEUR] AND NOT m_Input_PRG_MOUVEMENT_PS.CONF_Rotation[m_Input_INDEX_MOTEUR]) OR m_Input_MOTEUR.CONF_Mvt_Lineaire, input disabled if: (NOT PRG_User.ACTU_USER.MAINTENANCE AND m_Input_MOTEUR.MANUAL) OR (NOT PRG_User.ACTU_USER.FONCTION_SA AND NOT m_Input_MOTEUR.MANUAL)
        OnMouseClick: write the text variable via VisuDialogs.Numpad, min m_Input_PRG_MOUVEMENT_PS.CONF_MIN_SPEED[m_Input_INDEX_MOTEUR], max m_Input_PRG_MOUVEMENT_PS.CONF_MAX_SPEED[m_Input_INDEX_MOTEUR]
    RoundedRectangle (206,320 120x30), "%3.1f °", text variable: m_Input_MOTEUR.PRM_Position, invisible if: (NOT m_Input_PRG_MOUVEMENT_PS.CONF_Balayage[m_Input_INDEX_MOTEUR] AND NOT m_Input_PRG_MOUVEMENT_PS.CONF_Positionnement[m_Input_INDEX_MOTEUR]) OR m_Input_MOTEUR.CONF_Mvt_Lineaire, input disabled if: (NOT PRG_User.ACTU_USER.MAINTENANCE AND m_Input_MOTEUR.MANUAL) OR (NOT PRG_User.ACTU_USER.FONCTION_SA AND NOT m_Input_MOTEUR.MANUAL)
        OnMouseClick: write the text variable via VisuDialogs.Numpad, min m_Input_PRG_MOUVEMENT_PS.CONF_MIN_POS[m_Input_INDEX_MOTEUR], max m_Input_PRG_MOUVEMENT_PS.CONF_MAX_POS[m_Input_INDEX_MOTEUR]
    RoundedRectangle (206,356 120x30), "%3.1f °", text variable: m_Input_MOTEUR.PRM_Angle_Bal, invisible if: NOT m_Input_PRG_MOUVEMENT_PS.CONF_Balayage[m_Input_INDEX_MOTEUR] OR m_Input_MOTEUR.CONF_Mvt_Lineaire, input disabled if: (NOT PRG_User.ACTU_USER.MAINTENANCE AND m_Input_MOTEUR.MANUAL) OR (NOT PRG_User.ACTU_USER.FONCTION_SA AND NOT m_Input_MOTEUR.MANUAL)
        OnMouseClick: write the text variable via VisuDialogs.Numpad, min 0, max 360
END_VISUALIZATION

// ---- Visualizations/Symbole/MOUVEMENTS PS/AXE STD1/FCT_Part/VISU_AXE_STD1_ROT_ABS_FCT_ETAT.TcVIS
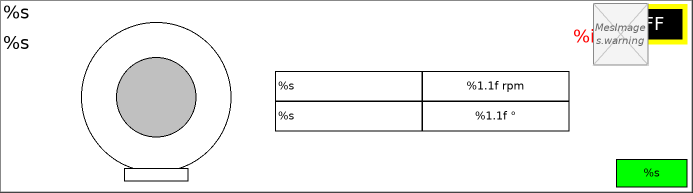
VISUALIZATION VISU_AXE_STD1_ROT_ABS_FCT_ETAT  // 693x193
VAR_IN_OUT
	m_Input_MOTEUR: BLOCK_AXE_STD1;
	m_Input_PRG_MOUVEMENT_PS: BLOCK_PRG_MOUVEMENT_PS;
END_VAR
VAR_INPUT CONSTANT
	m_Input_ID_NOM_XML : INT;
	m_Input_INDEX_MOTEUR : INT;
END_VAR
    Rectangle (0,0 693x193), "%s", text list: 'TextList_Type_Moteur', text index: m_Input_ID_NOM_XML
    Rectangle (0,28 107x30), "%s", text variable: m_Input_MOTEUR.MNEMO
    RoundedRectangle (275,71 147x30), "%s", text list: 'TextList_Moteurs', text index: 7
    RoundedRectangle (275,101 147x30), "%s", text list: 'TextList_Moteurs', text index: 12
    RoundedRectangle (422,71 147x30), "%1.1f rpm", text variable: m_Input_MOTEUR.STATE_Vit
    RoundedRectangle (422,101 147x30), "%1.1f °", text variable: m_Input_MOTEUR.STATE_Pos360
    Group (81,22 150x150)
        Ellipse (0,0 150x150)
        Ellipse (96,53 43x45), invisible if: m_Input_PRG_MOUVEMENT_PS.CONF_NB_REF[m_Input_INDEX_MOTEUR]<5
            p2277200375: m_Input_PRG_MOUVEMENT_PS.PRM_POS_REF[m_Input_INDEX_MOTEUR,5] + 90
        Ellipse (96,53 43x45), invisible if: m_Input_PRG_MOUVEMENT_PS.CONF_NB_REF[m_Input_INDEX_MOTEUR]<6
            p2277200375: m_Input_PRG_MOUVEMENT_PS.PRM_POS_REF[m_Input_INDEX_MOTEUR,6] + 90
        Ellipse (96,53 43x45), invisible if: m_Input_PRG_MOUVEMENT_PS.CONF_NB_REF[m_Input_INDEX_MOTEUR]<1
            p2277200375: m_Input_PRG_MOUVEMENT_PS.PRM_POS_REF[m_Input_INDEX_MOTEUR,1] + 90
        Ellipse (96,53 43x45), invisible if: m_Input_PRG_MOUVEMENT_PS.CONF_NB_REF[m_Input_INDEX_MOTEUR]<2
            p2277200375: m_Input_PRG_MOUVEMENT_PS.PRM_POS_REF[m_Input_INDEX_MOTEUR,2] + 90
        Ellipse (96,53 43x45), invisible if: m_Input_PRG_MOUVEMENT_PS.CONF_NB_REF[m_Input_INDEX_MOTEUR]<3
            p2277200375: m_Input_PRG_MOUVEMENT_PS.PRM_POS_REF[m_Input_INDEX_MOTEUR,3] + 90
        Ellipse (96,53 43x45), invisible if: m_Input_PRG_MOUVEMENT_PS.CONF_NB_REF[m_Input_INDEX_MOTEUR]<4
            p2277200375: m_Input_PRG_MOUVEMENT_PS.PRM_POS_REF[m_Input_INDEX_MOTEUR,4] + 90
        Ellipse (96,53 43x45), "4", invisible if: m_Input_PRG_MOUVEMENT_PS.CONF_NB_POSTE[m_Input_INDEX_MOTEUR]<4
            p2277200375: m_Input_MOTEUR.STATE_Pos360+ m_Input_PRG_MOUVEMENT_PS.PRM_POS_POSTE[m_Input_INDEX_MOTEUR,4] + 90
        Ellipse (96,53 43x45), "1", invisible if: m_Input_PRG_MOUVEMENT_PS.CONF_NB_POSTE[m_Input_INDEX_MOTEUR]<1
            p2277200375: m_Input_MOTEUR.STATE_Pos360 + m_Input_PRG_MOUVEMENT_PS.PRM_POS_POSTE[m_Input_INDEX_MOTEUR,1] + 90
        Ellipse (96,53 43x45), "2", invisible if: m_Input_PRG_MOUVEMENT_PS.CONF_NB_POSTE[m_Input_INDEX_MOTEUR]<2
            p2277200375: m_Input_MOTEUR.STATE_Pos360 + m_Input_PRG_MOUVEMENT_PS.PRM_POS_POSTE[m_Input_INDEX_MOTEUR,2] + 90
        Ellipse (96,53 43x45), "3", invisible if: m_Input_PRG_MOUVEMENT_PS.CONF_NB_POSTE[m_Input_INDEX_MOTEUR]<3
            p2277200375: m_Input_MOTEUR.STATE_Pos360 + m_Input_PRG_MOUVEMENT_PS.PRM_POS_POSTE[m_Input_INDEX_MOTEUR,3] + 90
    Group (81,22 150x150), invisible if: NOT m_Input_PRG_MOUVEMENT_PS.CONF_Poste_Central[m_Input_INDEX_MOTEUR]
        Ellipse (0,0 150x150)
        Ellipse (35,35 80x80)
    Rectangle (124,168 64x13)
    RoundedRectangle (607,4 80x40), invisible if: NOT m_Input_MOTEUR.OP_Validation.OK
    RoundedRectangle (607,4 80x40), invisible if: NOT m_Input_MOTEUR.OP_Validation.AR
    RoundedRectangle (607,4 80x40), invisible if: NOT m_Input_MOTEUR.OP_Validation.EC
    RoundedRectangle (612,9 70x30), "ON", invisible if: m_Input_MOTEUR.STATE_Ar
    RoundedRectangle (612,9 70x30), "OFF", invisible if: NOT m_Input_MOTEUR.STATE_Ar
    Rectangle (531,24 67x21), "%i", text variable: m_Input_MOTEUR.STATE_Err, invisible if: NOT m_Input_MOTEUR.STATE_NOK
    Image (593,3 55x62), invisible if: NOT m_Input_MOTEUR.STATE_NOK, image: MesImages.warning
    RoundedRectangle (616,159 71x28), "%s", invisible if: m_Input_MOTEUR.STATE_Homed OR m_Input_MOTEUR.CONF_No_Ref, text list: 'TextList_Moteurs', text index: 11
    RoundedRectangle (616,159 71x28), "%s", invisible if: NOT m_Input_MOTEUR.STATE_Homed OR m_Input_MOTEUR.CONF_No_Ref, text list: 'TextList_Moteurs', text index: 11
END_VISUALIZATION

// ---- Visualizations/Symbole/MOUVEMENTS PS/AXE STD1/FCT_Part/VISU_AXE_STD1_ROT_ABS_FCT_ETAT_OSC.TcVIS
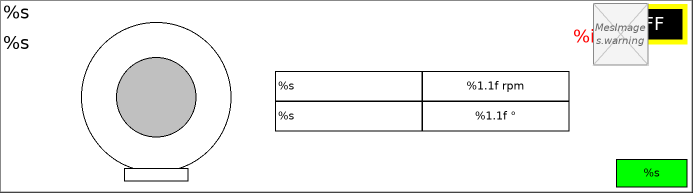
VISUALIZATION VISU_AXE_STD1_ROT_ABS_FCT_ETAT_OSC  // 693x193
VAR_IN_OUT
	m_Input_MOTEUR: BLOCK_AXE_STD1_OSCILLANT;
	m_Input_PRG_MOUVEMENT_PS: BLOCK_PRG_MOUVEMENT_PS;
END_VAR
VAR_INPUT CONSTANT
	m_Input_ID_NOM_XML : INT;
	m_Input_INDEX_MOTEUR : INT;
END_VAR
    Rectangle (0,0 693x193), "%s", text list: 'TextList_Type_Moteur', text index: m_Input_ID_NOM_XML
    Rectangle (0,28 107x30), "%s", text variable: m_Input_MOTEUR.MNEMO
    RoundedRectangle (275,71 147x30), "%s", text list: 'TextList_Moteurs', text index: 7
    RoundedRectangle (275,101 147x30), "%s", text list: 'TextList_Moteurs', text index: 12
    RoundedRectangle (422,71 147x30), "%1.1f rpm", text variable: m_Input_MOTEUR.STATE_Vit
    RoundedRectangle (422,101 147x30), "%1.1f °", text variable: m_Input_MOTEUR.STATE_Pos
    Group (81,22 150x150), invisible if: NOT m_Input_PRG_MOUVEMENT_PS.CONF_Poste_Central[m_Input_INDEX_MOTEUR]
        Ellipse (0,0 150x150)
        Ellipse (35,35 80x80)
    Rectangle (124,168 64x13)
    RoundedRectangle (607,4 80x40), invisible if: NOT m_Input_MOTEUR.OP_Validation.OK
    RoundedRectangle (607,4 80x40), invisible if: NOT m_Input_MOTEUR.OP_Validation.AR
    RoundedRectangle (607,4 80x40), invisible if: NOT m_Input_MOTEUR.OP_Validation.EC
    RoundedRectangle (612,9 70x30), "ON", invisible if: m_Input_MOTEUR.STATE_Ar
    RoundedRectangle (612,9 70x30), "OFF", invisible if: NOT m_Input_MOTEUR.STATE_Ar
    Rectangle (531,24 67x21), "%i", text variable: m_Input_MOTEUR.STATE_Err, invisible if: NOT m_Input_MOTEUR.STATE_NOK
    Image (593,3 55x62), invisible if: NOT m_Input_MOTEUR.STATE_NOK, image: MesImages.warning
    RoundedRectangle (616,159 71x28), "%s", invisible if: m_Input_MOTEUR.STATE_Homed OR m_Input_MOTEUR.CONF_No_Ref, text list: 'TextList_Moteurs', text index: 11
    RoundedRectangle (616,159 71x28), "%s", invisible if: NOT m_Input_MOTEUR.STATE_Homed OR m_Input_MOTEUR.CONF_No_Ref, text list: 'TextList_Moteurs', text index: 11
END_VISUALIZATION

// ---- Visualizations/Symbole/MOUVEMENTS PS/AXE STD1/VISU_AXE_STD1_LIN_REL.TcVIS
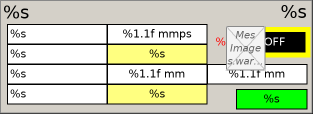
VISUALIZATION VISU_AXE_STD1_LIN_REL  // 313x114
VAR_IN_OUT
	m_Input_MOTEUR: BLOCK_AXE_STD1;
	m_Input_PRG_MOUVEMENT_PS: BLOCK_PRG_MOUVEMENT_PS;
END_VAR
VAR_Input
	m_Input_ID_NOM_XML : INT;
	m_Input_INDEX_MOTEUR : INT;
	m_Input_Ref_Trf:	INT;
	m_Input_NumFrame_Manu:	USINT;		(*numéro de frame à afficher dans le synoptique MANUEL*)
END_VAR
    Rectangle (0,0 313x114), "%s", text list: 'TextList_Type_Moteur', text index: m_Input_ID_NOM_XML
    Rectangle (223,4 87x16), "%s", text variable: m_Input_MOTEUR.MNEMO
    RoundedRectangle (7,24 100x20), "%s", text list: 'TextList_Moteurs', text index: 7
    RoundedRectangle (7,44 100x20), "%s", text list: 'TextList_Moteurs', text index: 8
    RoundedRectangle (7,64 100x20), "%s", text list: 'TextList_Moteurs', text index: 9
    RoundedRectangle (7,84 100x20), "%s", text list: 'TextList_Moteurs', text index: 10
    RoundedRectangle (107,24 100x20), "%1.1f mmps", text variable: m_Input_MOTEUR.STATE_Vit
    RoundedRectangle (107,44 100x20), "%s", text variable: m_Input_MOTEUR.CONF_ID_POSTE[m_Input_MOTEUR.PRM_NPOSTE]
    RoundedRectangle (107,64 100x20), "%1.1f mm", text variable: m_Input_MOTEUR.STATE_Pos_Rel
    RoundedRectangle (207,64 100x20), "%1.1f mm", text variable: m_Input_MOTEUR.STATE_Pos
    RoundedRectangle (107,84 100x20), "%s", text variable: m_Input_MOTEUR.CONF_ID_REF[m_Input_MOTEUR.PRM_NRef]
    RoundedRectangle (236,89 71x20), "%s", invisible if: m_Input_MOTEUR.STATE_Homed OR m_Input_MOTEUR.CONF_No_Ref, text list: 'TextList_Moteurs', text index: 11
    RoundedRectangle (236,89 71x20), "%s", invisible if: NOT m_Input_MOTEUR.STATE_Homed OR m_Input_MOTEUR.CONF_No_Ref, text list: 'TextList_Moteurs', text index: 11
    RoundedRectangle (240,27 70x30), invisible if: NOT m_Input_MOTEUR.OP_Validation.OK
    RoundedRectangle (240,27 70x30), invisible if: NOT m_Input_MOTEUR.OP_Validation.AR
    RoundedRectangle (240,27 70x30), invisible if: NOT m_Input_MOTEUR.OP_Validation.EC
    RoundedRectangle (245,32 60x20), "ON", invisible if: m_Input_MOTEUR.STATE_Ar
    RoundedRectangle (245,32 60x20), "OFF", invisible if: NOT m_Input_MOTEUR.STATE_Ar
    Rectangle (165,34 67x21), "%i", text variable: m_Input_MOTEUR.STATE_Err, invisible if: NOT m_Input_MOTEUR.STATE_NOK
    Image (226,26 39x44), invisible if: NOT m_Input_MOTEUR.STATE_NOK, image: MesImages.warning
    Rectangle (0,0 313x114)
        OnMouseClick: execute { .VISU_INDEX_MANU := m_Input_NumFrame_Manu; }
        OnMouseClick: change screen: SYN_MANUEL
END_VISUALIZATION

// ---- Visualizations/Symbole/MOUVEMENTS PS/AXE STD1/VISU_AXE_STD1_MANU.TcVIS
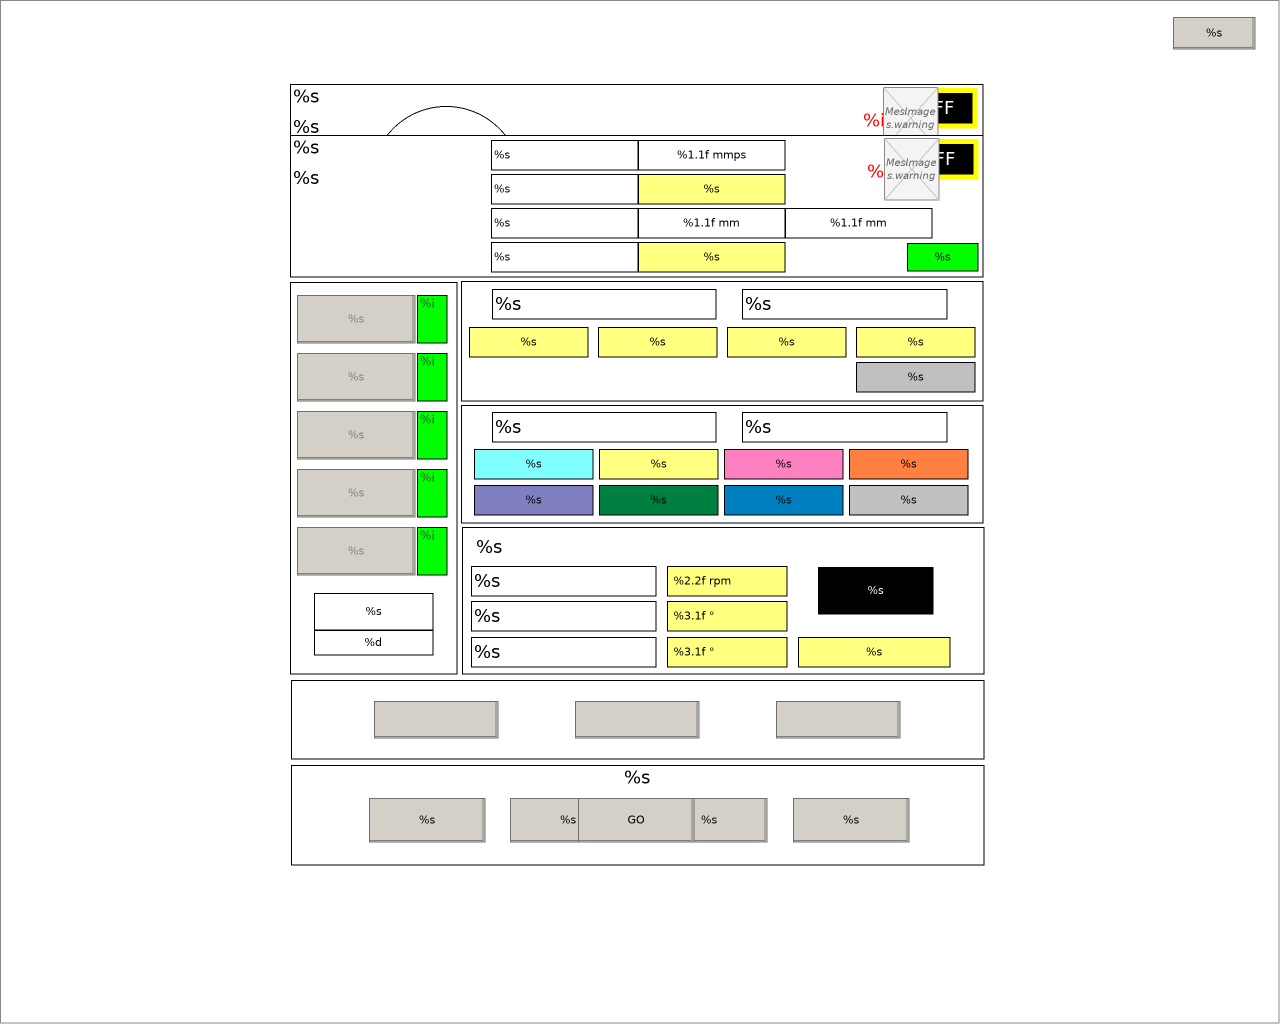
VISUALIZATION VISU_AXE_STD1_MANU  // 1280x1024
VAR_IN_OUT
	m_Input_MOTEUR: BLOCK_AXE_STD1;
	m_Input_PRG_MOUVEMENT_PS: BLOCK_PRG_MOUVEMENT_PS;
END_VAR
VAR_INPUT
	m_Input_ID_NOM_XML : INT;
	m_Input_INDEX_MOTEUR : INT;
	m_Input_Ref_Trf:	USINT;
END_VAR
    Frame (290,84 696x199), invisible if: NOT m_Input_PRG_MOUVEMENT_PS.CONF_ROT_ABS[m_Input_INDEX_MOTEUR]
        shows VISU_AXE_STD1_ROT_ABS_FCT_ETAT(m_Input_MOTEUR := m_Input_MOTEUR, m_Input_PRG_MOUVEMENT_PS := m_Input_PRG_MOUVEMENT_PS, m_Input_ID_NOM_XML := m_Input_ID_NOM_XML, m_Input_INDEX_MOTEUR := m_Input_INDEX_MOTEUR)
    Button (1173,17 82x32), "%s", text list: 'TextList_Basiques', text index: 8
        OnMouseClick: change screen: Previous 
        OnMouseClick: execute { .VISU_INDEX_MANU := 0; }
    Frame (290,135 694x145), invisible if: NOT m_Input_PRG_MOUVEMENT_PS.CONF_LIN_REL[m_Input_INDEX_MOTEUR]
        shows VISU_AXE_STD1_LIN_REL_FCT_ETAT(m_Input_MOTEUR := m_Input_MOTEUR, m_Input_PRG_MOUVEMENT_PS := m_Input_PRG_MOUVEMENT_PS, m_Input_ID_NOM_XML := m_Input_ID_NOM_XML)
        p625233746: m_Input_MOTEUR
        p171577005: m_Input_PRG_MOUVEMENT_PS
        p3150284580: m_Input_ID_NOM_XML
    Frame (288,283 169x397)
        shows VISU_AXE_STD1_FCT_OP(m_Input_MOTEUR := m_Input_MOTEUR, m_Input_PRG_MOUVEMENT_PS := m_Input_PRG_MOUVEMENT_PS, m_Input_INDEX_MOTEUR := m_Input_INDEX_MOTEUR)
    Frame (461,281 524x460), invisible if: NOT m_Input_PRG_MOUVEMENT_PS.CONF_LIN_REL[m_Input_INDEX_MOTEUR] AND NOT m_Input_PRG_MOUVEMENT_PS.CONF_ROT_ABS[m_Input_INDEX_MOTEUR]
        shows VISU_AXE_STD1_LIN_ROT_FCT_CONS(m_Input_MOTEUR := m_Input_MOTEUR, m_Input_PRG_MOUVEMENT_PS := m_Input_PRG_MOUVEMENT_PS, m_Input_INDEX_MOTEUR := m_Input_INDEX_MOTEUR)
    Frame (291,680 700x79)
        shows VISU_AXE_STD1_FCT_MANU(m_Input_MOTEUR := m_Input_MOTEUR, m_Input_PRG_MOUVEMENT_PS := m_Input_PRG_MOUVEMENT_PS, m_Input_INDEX_MOTEUR := m_Input_INDEX_MOTEUR)
    Frame (291,765 695x105), invisible if: NOT m_Input_PRG_MOUVEMENT_PS.CONF_TRF[m_Input_INDEX_MOTEUR]
        shows VISU_AXE_STD1_FCT_TRF(m_Input_MOTEUR := m_Input_MOTEUR, m_Input_PRG_MOUVEMENT_PS := m_Input_PRG_MOUVEMENT_PS, m_Input_INDEX_MOTEUR := m_Input_INDEX_MOTEUR, m_Input_Ref_Trf := m_Input_REF_TRF)
        pReferences[0]: m_Input_REF_TRF=m_Input_REF_TRF
END_VISUALIZATION

// ---- Visualizations/Symbole/MOUVEMENTS PS/AXE STD1/VISU_AXE_STD1_MANU_OSC.TcVIS
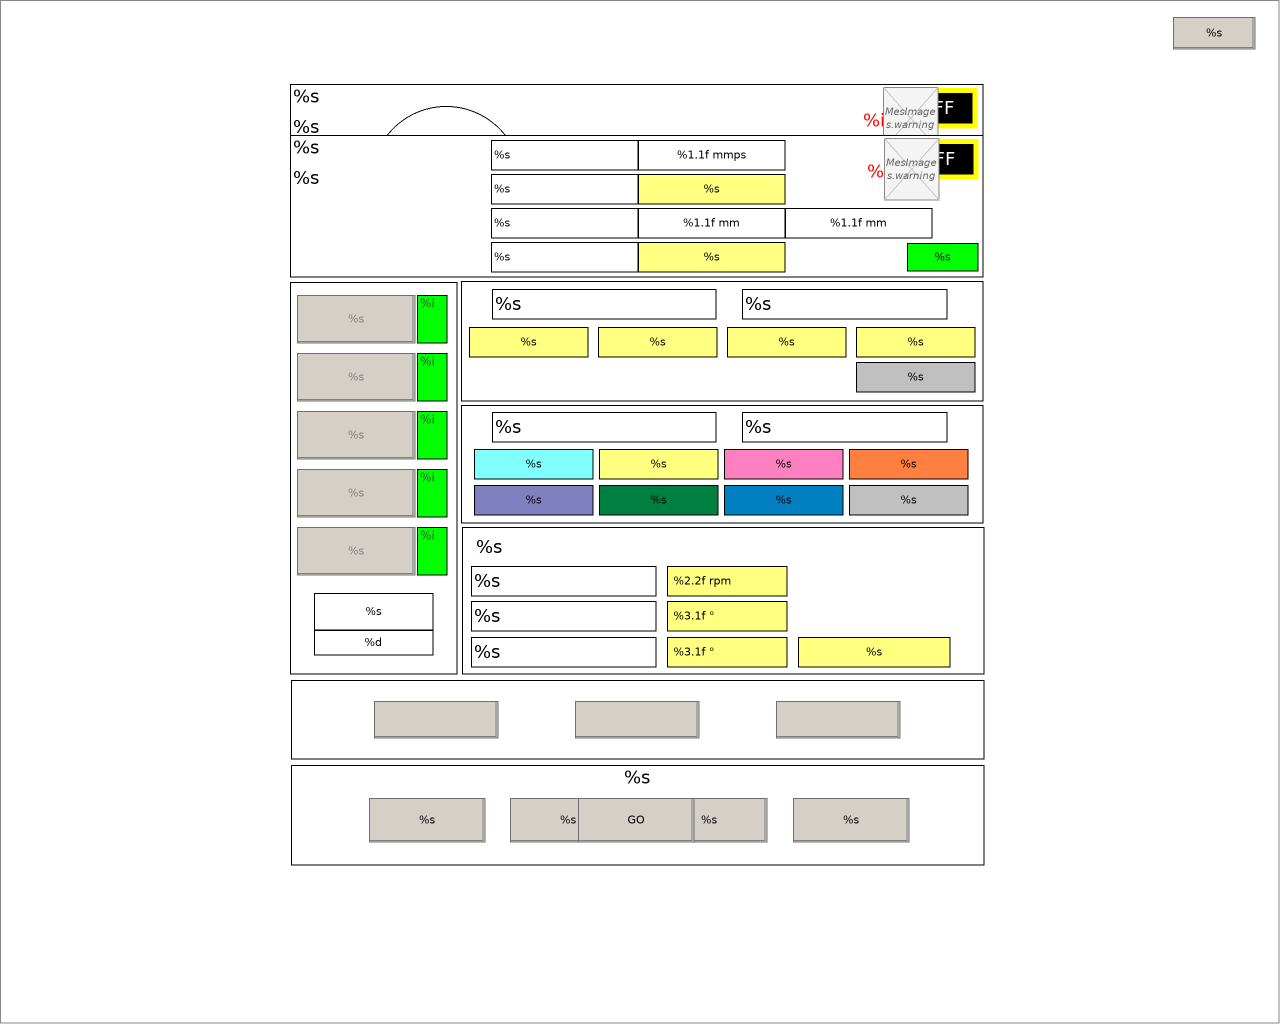
VISUALIZATION VISU_AXE_STD1_MANU_OSC  // 1280x1024
VAR_IN_OUT
	m_Input_MOTEUR: BLOCK_AXE_STD1_OSCILLANT;
	m_Input_PRG_MOUVEMENT_PS: BLOCK_PRG_MOUVEMENT_PS;
END_VAR
VAR_INPUT
	m_Input_ID_NOM_XML : INT;
	m_Input_INDEX_MOTEUR : INT;
	m_Input_Ref_Trf:	USINT;
END_VAR
    Frame (290,84 696x199), invisible if: NOT m_Input_PRG_MOUVEMENT_PS.CONF_ROT_ABS[m_Input_INDEX_MOTEUR]
        shows VISU_AXE_STD1_ROT_ABS_FCT_ETAT_OSC(m_Input_MOTEUR := m_Input_MOTEUR, m_Input_PRG_MOUVEMENT_PS := m_Input_PRG_MOUVEMENT_PS, m_Input_ID_NOM_XML := m_Input_ID_NOM_XML, m_Input_INDEX_MOTEUR := m_Input_INDEX_MOTEUR)
        p625233746: m_Input_MOTEUR
        p171577005: m_Input_PRG_MOUVEMENT_PS
        p3150284580: m_Input_ID_NOM_XML
        p114361821: m_Input_INDEX_MOTEUR
    Button (1173,17 82x32), "%s", text list: 'TextList_Basiques', text index: 8
        OnMouseClick: change screen: Previous 
        OnMouseClick: execute { .VISU_INDEX_MANU := 0; }
    Frame (290,135 694x145), invisible if: NOT m_Input_PRG_MOUVEMENT_PS.CONF_LIN_REL[m_Input_INDEX_MOTEUR]
        shows VISU_AXE_STD1_LIN_REL_FCT_ETAT_OSC(m_Input_MOTEUR := m_Input_MOTEUR, m_Input_PRG_MOUVEMENT_PS := m_Input_PRG_MOUVEMENT_PS, m_Input_ID_NOM_XML := m_Input_ID_NOM_XML)
        p625233746: m_Input_MOTEUR
        p171577005: m_Input_PRG_MOUVEMENT_PS
        p3150284580: m_Input_ID_NOM_XML
    Frame (288,283 169x397)
        shows VISU_AXE_STD1_FCT_OP_OSC(m_Input_MOTEUR := m_Input_MOTEUR, m_Input_PRG_MOUVEMENT_PS := m_Input_PRG_MOUVEMENT_PS, m_Input_INDEX_MOTEUR := m_Input_INDEX_MOTEUR)
        p625233746: m_Input_MOTEUR
        p171577005: m_Input_PRG_MOUVEMENT_PS
        p114361821: m_Input_INDEX_MOTEUR
    Frame (461,281 524x460), invisible if: NOT m_Input_PRG_MOUVEMENT_PS.CONF_LIN_REL[m_Input_INDEX_MOTEUR] AND NOT m_Input_PRG_MOUVEMENT_PS.CONF_ROT_ABS[m_Input_INDEX_MOTEUR]
        shows VISU_AXE_STD1_LIN_ROT_FCT_CONS_OSC(m_Input_MOTEUR := m_Input_MOTEUR, m_Input_PRG_MOUVEMENT_PS := m_Input_PRG_MOUVEMENT_PS, m_Input_INDEX_MOTEUR := m_Input_INDEX_MOTEUR)
        p625233746: m_Input_MOTEUR
        p171577005: m_Input_PRG_MOUVEMENT_PS
        p114361821: m_Input_INDEX_MOTEUR
    Frame (291,680 700x79)
        shows VISU_AXE_STD1_FCT_MANU_OSC(m_Input_MOTEUR := m_Input_MOTEUR, m_Input_PRG_MOUVEMENT_PS := m_Input_PRG_MOUVEMENT_PS, m_Input_INDEX_MOTEUR := m_Input_INDEX_MOTEUR)
        p625233746: m_Input_MOTEUR
        p171577005: m_Input_PRG_MOUVEMENT_PS
        p114361821: m_Input_INDEX_MOTEUR
    Frame (291,765 695x105), invisible if: NOT m_Input_PRG_MOUVEMENT_PS.CONF_TRF[m_Input_INDEX_MOTEUR]
        shows VISU_AXE_STD1_FCT_TRF_OSC(m_Input_MOTEUR := m_Input_MOTEUR, m_Input_PRG_MOUVEMENT_PS := m_Input_PRG_MOUVEMENT_PS, m_Input_INDEX_MOTEUR := m_Input_INDEX_MOTEUR, m_Input_Ref_Trf := m_Input_REF_TRF)
        p625233746: m_Input_MOTEUR
        p171577005: m_Input_PRG_MOUVEMENT_PS
        p114361821: m_Input_INDEX_MOTEUR
        p3023144840: m_Input_REF_TRF
END_VISUALIZATION

// ---- Visualizations/Symbole/MOUVEMENTS PS/AXE STD1/VISU_AXE_STD1_ROT_ABS.TcVIS
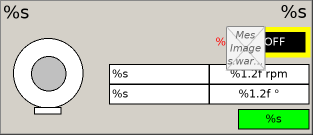
VISUALIZATION VISU_AXE_STD1_ROT_ABS  // 313x135
VAR_IN_OUT
	m_Input_MOTEUR: BLOCK_AXE_STD1;
	m_Input_PRG_MOUVEMENT_PS: BLOCK_PRG_MOUVEMENT_PS;
END_VAR
VAR_Input
	m_Input_ID_NOM_XML : INT;
	m_Input_INDEX_MOTEUR : INT;
	m_Input_Ref_Trf:	INT;
	m_Input_NumFrame_Manu:	USINT;		(*numéro de frame à afficher dans le synoptique MANUEL*)
END_VAR
    Rectangle (0,0 313x135), "%s", text list: 'TextList_Type_Moteur', text index: m_Input_ID_NOM_XML
    Rectangle (223,4 87x16), "%s", text variable: m_Input_MOTEUR.MNEMO
    RoundedRectangle (109,64 100x20), "%s", text list: 'TextList_Moteurs', text index: 7
    RoundedRectangle (109,84 100x20), "%s", text list: 'TextList_Moteurs', text index: 9
    RoundedRectangle (209,64 100x20), "%1.2f rpm", text variable: m_Input_MOTEUR.STATE_Vit
    RoundedRectangle (209,84 100x20), "%1.2f °", text variable: m_Input_MOTEUR.STATE_Pos360
    RoundedRectangle (238,109 71x20), "%s", invisible if: m_Input_MOTEUR.STATE_Homed OR m_Input_MOTEUR.CONF_No_Ref, text list: 'TextList_Moteurs', text index: 11
    RoundedRectangle (238,109 71x20), "%s", invisible if: NOT m_Input_MOTEUR.STATE_Homed OR m_Input_MOTEUR.CONF_No_Ref, text list: 'TextList_Moteurs', text index: 11
    RoundedRectangle (240,27 70x30), invisible if: NOT m_Input_MOTEUR.OP_Validation.OK
    RoundedRectangle (240,27 70x30), invisible if: NOT m_Input_MOTEUR.OP_Validation.AR
    RoundedRectangle (240,27 70x30), invisible if: NOT m_Input_MOTEUR.OP_Validation.EC
    RoundedRectangle (245,32 60x20), "ON", invisible if: m_Input_MOTEUR.STATE_Ar
    RoundedRectangle (245,32 60x20), "OFF", invisible if: NOT m_Input_MOTEUR.STATE_Ar
    Rectangle (165,34 67x21), "%i", text variable: m_Input_MOTEUR.STATE_Err, invisible if: NOT m_Input_MOTEUR.STATE_NOK
    Image (226,26 39x44), invisible if: NOT m_Input_MOTEUR.STATE_NOK, image: MesImages.warning
    Rectangle (0,0 313x135)
        OnMouseClick: execute { .VISU_INDEX_MANU := m_Input_NumFrame_Manu; }
        OnMouseClick: change screen: SYN_MANUEL
    Ellipse (13,38 70x70)
    Ellipse (58,63 20x20), invisible if: m_Input_PRG_MOUVEMENT_PS.CONF_NB_REF[m_Input_INDEX_MOTEUR]<2
        p2277200375: m_Input_PRG_MOUVEMENT_PS.PRM_POS_REF[m_Input_INDEX_MOTEUR,2] + 90
    Ellipse (58,63 20x20), invisible if: m_Input_PRG_MOUVEMENT_PS.CONF_NB_REF[m_Input_INDEX_MOTEUR]<3
        p2277200375: m_Input_PRG_MOUVEMENT_PS.PRM_POS_REF[m_Input_INDEX_MOTEUR,3] + 90
    Ellipse (58,63 20x20), invisible if: m_Input_PRG_MOUVEMENT_PS.CONF_NB_REF[m_Input_INDEX_MOTEUR]<4
        p2277200375: m_Input_PRG_MOUVEMENT_PS.PRM_POS_REF[m_Input_INDEX_MOTEUR,4] + 90
    Ellipse (58,63 20x20), invisible if: m_Input_PRG_MOUVEMENT_PS.CONF_NB_REF[m_Input_INDEX_MOTEUR]<5
        p2277200375: m_Input_PRG_MOUVEMENT_PS.PRM_POS_REF[m_Input_INDEX_MOTEUR,5] + 90
    Ellipse (58,63 20x20), invisible if: m_Input_PRG_MOUVEMENT_PS.CONF_NB_REF[m_Input_INDEX_MOTEUR]<6
        p2277200375: m_Input_PRG_MOUVEMENT_PS.PRM_POS_REF[m_Input_INDEX_MOTEUR,6] + 90
    Ellipse (58,63 20x20), invisible if: m_Input_PRG_MOUVEMENT_PS.CONF_NB_REF[m_Input_INDEX_MOTEUR]<1
        p2277200375: m_Input_PRG_MOUVEMENT_PS.PRM_POS_REF[m_Input_INDEX_MOTEUR,1] + 90
    Ellipse (58,63 20x20), "1", invisible if: m_Input_PRG_MOUVEMENT_PS.CONF_NB_POSTE[m_Input_INDEX_MOTEUR]<1
        p2277200375: m_Input_MOTEUR.STATE_Pos360 + m_Input_PRG_MOUVEMENT_PS.PRM_POS_POSTE[m_Input_INDEX_MOTEUR,1] + 90
    Ellipse (58,63 20x20), "2", invisible if: m_Input_PRG_MOUVEMENT_PS.CONF_NB_POSTE[m_Input_INDEX_MOTEUR]<2
        p2277200375: m_Input_MOTEUR.STATE_Pos360 + m_Input_PRG_MOUVEMENT_PS.PRM_POS_POSTE[m_Input_INDEX_MOTEUR,2] + 90
    Ellipse (58,63 20x20), "3", invisible if: m_Input_PRG_MOUVEMENT_PS.CONF_NB_POSTE[m_Input_INDEX_MOTEUR]<3
        p2277200375: m_Input_MOTEUR.STATE_Pos360 + m_Input_PRG_MOUVEMENT_PS.PRM_POS_POSTE[m_Input_INDEX_MOTEUR,3] + 90
    Ellipse (58,63 20x20), "4", invisible if: m_Input_PRG_MOUVEMENT_PS.CONF_NB_POSTE[m_Input_INDEX_MOTEUR]<4
        p2277200375: m_Input_MOTEUR.STATE_Pos360 + m_Input_PRG_MOUVEMENT_PS.PRM_POS_POSTE[m_Input_INDEX_MOTEUR,4] + 90
    Group (13,38 70x70), invisible if: NOT m_Input_PRG_MOUVEMENT_PS.CONF_Poste_Central[m_Input_INDEX_MOTEUR]
        Ellipse (0,0 70x70)
        Ellipse (18,18 35x35)
    Rectangle (34,107 27x7)
END_VISUALIZATION

// ---- Visualizations/Symbole/MOUVEMENTS PS/AXE STD1/VISU_AXE_STD1_ROT_ABS_OSC.TcVIS
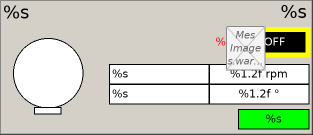
VISUALIZATION VISU_AXE_STD1_ROT_ABS_OSC  // 313x135
VAR_IN_OUT
	m_Input_MOTEUR: BLOCK_AXE_STD1_OSCILLANT;
	m_Input_PRG_MOUVEMENT_PS: BLOCK_PRG_MOUVEMENT_PS;
END_VAR
VAR_Input
	m_Input_ID_NOM_XML : INT;
	m_Input_INDEX_MOTEUR : INT;
	m_Input_Ref_Trf:	INT;
	m_Input_NumFrame_Manu:	USINT;		(*numéro de frame à afficher dans le synoptique MANUEL*)
END_VAR
    Rectangle (0,0 313x135), "%s", text list: 'TextList_Type_Moteur', text index: m_Input_ID_NOM_XML
    Rectangle (223,4 87x16), "%s", text variable: m_Input_MOTEUR.MNEMO
    RoundedRectangle (109,64 100x20), "%s", text list: 'TextList_Moteurs', text index: 7
    RoundedRectangle (109,84 100x20), "%s", text list: 'TextList_Moteurs', text index: 9
    RoundedRectangle (209,64 100x20), "%1.2f rpm", text variable: m_Input_MOTEUR.STATE_Vit
    RoundedRectangle (209,84 100x20), "%1.2f °", text variable: m_Input_MOTEUR.STATE_Pos
    RoundedRectangle (238,109 71x20), "%s", invisible if: m_Input_MOTEUR.STATE_Homed OR m_Input_MOTEUR.CONF_No_Ref, text list: 'TextList_Moteurs', text index: 11
    RoundedRectangle (238,109 71x20), "%s", invisible if: NOT m_Input_MOTEUR.STATE_Homed OR m_Input_MOTEUR.CONF_No_Ref, text list: 'TextList_Moteurs', text index: 11
    RoundedRectangle (240,27 70x30), invisible if: NOT m_Input_MOTEUR.OP_Validation.OK
    RoundedRectangle (240,27 70x30), invisible if: NOT m_Input_MOTEUR.OP_Validation.AR
    RoundedRectangle (240,27 70x30), invisible if: NOT m_Input_MOTEUR.OP_Validation.EC
    RoundedRectangle (245,32 60x20), "ON", invisible if: m_Input_MOTEUR.STATE_Ar
    RoundedRectangle (245,32 60x20), "OFF", invisible if: NOT m_Input_MOTEUR.STATE_Ar
    Rectangle (165,34 67x21), "%i", text variable: m_Input_MOTEUR.STATE_Err, invisible if: NOT m_Input_MOTEUR.STATE_NOK
    Image (226,26 39x44), invisible if: NOT m_Input_MOTEUR.STATE_NOK, image: MesImages.warning
    Rectangle (0,0 313x135)
        OnMouseClick: execute { .VISU_INDEX_MANU := m_Input_NumFrame_Manu; }
        OnMouseClick: change screen: SYN_MANUEL
    Ellipse (13,38 70x70)
    Rectangle (34,107 27x7)
END_VISUALIZATION

// ---- Visualizations/Symbole/MOUVEMENTS PS/VISU_CANNE_TRANSFERT.TcVIS
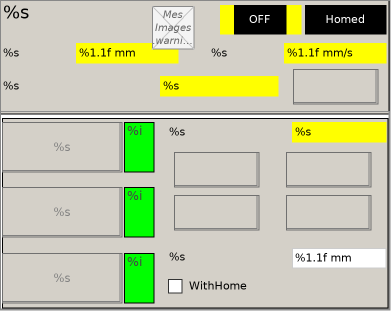
VISUALIZATION VISU_CANNE_TRANSFERT  // 391x311
VAR_IN_OUT
	m_Input_Moteur:				BLOCK_AXE_STD1;
	m_Input_Id_Poste:			INT;
	m_Input_Command_Visible:	BOOL;	
END_VAR
    Rectangle (0,0 389x114), "%s", text list: 'TextList_Canne_Transfert', text index: 0
    RoundedRectangle (220,5 81x29), invisible if: NOT m_Input_Moteur.OP_Validation.AR
    RoundedRectangle (220,5 81x29), invisible if: NOT m_Input_Moteur.OP_Validation.OK
    RoundedRectangle (220,5 81x29), invisible if: NOT m_Input_Moteur.OP_Validation.EC
    RoundedRectangle (234,5 52x29), "ON", invisible if: m_Input_Moteur.STATE_Ar
    RoundedRectangle (234,5 52x29), "OFF", invisible if: NOT m_Input_Moteur.STATE_Ar
    RoundedRectangle (305,5 81x29), "Homed", invisible if: NOT m_Input_Moteur.STATE_Homed OR m_Input_Moteur.CONF_No_Ref
    RoundedRectangle (305,5 81x29), "Homed", invisible if: m_Input_Moteur.STATE_Homed OR m_Input_Moteur.CONF_No_Ref
    Textfield (0,43 120x20), "%s", text list: 'TextList_Canne_Transfert', text index: 1
    Textfield (76,43 102x20), "%1.1f mm", text variable: m_Input_Moteur.STATE_Pos
    Textfield (208,43 120x20), "%s", text list: 'TextList_Canne_Transfert', text index: 2
    Textfield (284,43 102x20), "%1.1f mm/s", text variable: m_Input_Moteur.STATE_Vit
    Textfield (0,76 153x20), "%s", text list: 'TextList_Canne_Transfert', text index: 3
    Textfield (160,76 118x20), "%s", text list: 'TextList_Position_Canne', text index: m_Input_Id_Poste
    GroupBox (0,103 389x206), invisible if: NOT m_Input_Command_Visible
        Rectangle (2,15 386x190)
        Frame (2,19 152x49)
            shows VISU_FCTS_SA(m_Input_ID_XML := 6, m_Input_UserRight := PRG_USER.ACTU_USER.FONCTION_SA, m_Input_Operation := m_Input_Moteur.OP_Validation)
        Frame (2,150 152x49)
            shows VISU_FCTS_SA(m_Input_ID_XML := 8, m_Input_UserRight := PRG_USER.ACTU_USER.FONCTION_SA, m_Input_Operation := m_Input_Moteur.OP_Position)
        Frame (2,84 152x49)
            shows VISU_FCTS_SA(m_Input_ID_XML := 7, m_Input_UserRight := PRG_USER.ACTU_USER.FONCTION_SA, m_Input_Operation := m_Input_Moteur.OP_Stop)
        Checkbox (166,171 145x24), "WithHome", variable: m_Input_Moteur.PRM_GoToHome
        Textfield (166,19 120x20), "%s", text list: 'TextList_Canne_Transfert', text index: 4
        Textfield (292,19 94x20), "%s", text list: 'TextList_Position_Canne', text index: m_Input_Moteur.PRM_NRef
        Button (174,49 85x35), input disabled if: NOT PRG_USER.ACTU_USER.FONCTION_SA, text list: 'TextList_Position_Canne', text index: 0
            OnMouseClick: execute { m_Input_Moteur.PRM_NREF := 0; }
        Button (286,49 85x35), input disabled if: NOT PRG_USER.ACTU_USER.FONCTION_SA, text list: 'TextList_Position_Canne', text index: 1
            OnMouseClick: execute { m_Input_Moteur.PRM_NREF := 1; }
        Button (174,92 85x35), input disabled if: NOT PRG_USER.ACTU_USER.FONCTION_SA, text list: 'TextList_Position_Canne', text index: 2
            OnMouseClick: execute { m_Input_Moteur.PRM_NREF := 2; }
        Textfield (166,144 120x20), "%s", text list: 'TextList_Canne_Transfert', text index: 5
        Textfield (292,145 94x20), "%1.1f mm", text variable: m_Input_Moteur.PRM_Position
            OnMouseClick: write the text variable via VisuDialogs.NumpadExtended, min -100, max 100
        Button (286,92 85x35), input disabled if: NOT PRG_USER.ACTU_USER.FONCTION_SA, text list: 'TextList_Position_Canne', text index: 3
            OnMouseClick: execute { m_Input_Moteur.PRM_NREF := 3; }
    Button (293,69 85x35), text list: 'TextList_Canne_Transfert', text index: 7
        toggle m_Input_Command_Visible
    Image (152,6 42x43), invisible if: NOT m_Input_Moteur.STATE_NOK, image: MesImages.warning
END_VISUALIZATION

// ---- Visualizations/Symbole/MOUVEMENTS PS/VISU_CLAPET_V.TcVIS
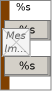
VISUALIZATION VISU_CLAPET_V  // 52x91
VAR_IN_OUT
	m_Input_CLAPET : BLOCK_ACTUATOR;
	m_Input_MAINT:		BOOL;
END_VAR
    Rectangle (0,0 9x89), invisible if: NOT m_Input_CLAPET.STATE_ON
    Rectangle (0,0 9x89), invisible if: (m_Input_CLAPET.STATE_ON OR m_Input_CLAPET.STATE_OFF) <> 0
    Rectangle (0,0 9x89), invisible if: NOT m_Input_CLAPET.STATE_OFF
    Rectangle (0,1 47x12), "%s", text variable: m_Input_CLAPET.MNEMO
    Button (4,20 46x20), "%s", invisible if: NOT m_Input_CLAPET.AUTOR_On_IHM OR NOT m_Input_MAINT, input disabled if: NOT m_Input_CLAPET.AUTOR_On_IHM OR NOT m_Input_MAINT, text list: 'TextList_Orders', text index: 0
        tap m_Input_CLAPET.M_On
    Button (4,56 46x20), "%s", invisible if: NOT m_Input_CLAPET.AUTOR_Off_IHM OR NOT m_Input_MAINT, input disabled if: NOT m_Input_CLAPET.AUTOR_Off_IHM OR NOT m_Input_MAINT, text list: 'TextList_Orders', text index: 1
        tap m_Input_CLAPET.M_Off
    Image (2,28 28x28), invisible if: NOT m_Input_CLAPET.STATE_NOK, image: MesImages.warning
END_VISUALIZATION

// ---- Visualizations/Symbole/MOUVEMENTS PS/VISU_CONFIG_POSITION_REF.TcVIS
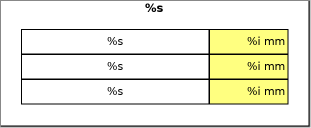
VISUALIZATION VISU_CONFIG_POSITION_REF  // 311x128
VAR_IN_OUT
	m_Input_Index:			INT;
END_VAR
    RoundedRectangle (0,0 309x126), "%s", text list: 'TextList_Config_Mouvements', text index: 2
    Rectangle (209,29 79x25), "%i mm", text variable: PRG_MOUVEMENT_PS.PRM_POS_REF[m_Input_Index,1], input disabled if: NOT Global_Variables.PRG_USER.ACTU_USER.CONF_MACHINE
        OnMouseDown: write the text variable via VisuDialogs.Numpad, min 0, max 900
    Rectangle (21,29 188x25), "%s", text list: 'TextList_Position_Canne', text index: 1
    Rectangle (21,54 188x25), "%s", text list: 'TextList_Position_Canne', text index: 2
    Rectangle (21,79 188x25), "%s", text list: 'TextList_Position_Canne', text index: 3
    Rectangle (209,54 79x25), "%i mm", text variable: PRG_MOUVEMENT_PS.PRM_POS_REF[m_Input_Index,2], input disabled if: NOT Global_Variables.PRG_USER.ACTU_USER.CONF_MACHINE
        OnMouseDown: write the text variable via VisuDialogs.Numpad, min 0, max 900
    Rectangle (209,79 79x25), "%i mm", text variable: PRG_MOUVEMENT_PS.PRM_POS_REF[m_Input_Index,3], input disabled if: NOT Global_Variables.PRG_USER.ACTU_USER.CONF_MACHINE
        OnMouseDown: write the text variable via VisuDialogs.Numpad, min 0, max 900
END_VISUALIZATION

// ---- Visualizations/Symbole/MOUVEMENTS PS/VISU_ROT.TcVIS
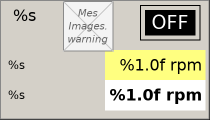
VISUALIZATION VISU_ROT  // 210x120
VAR_IN_OUT
	m_Input_ROT:		BLOCK_ROTATION_CONTINUE_ATV;
END_VAR
    RoundedRectangle (0,0 210x120)
    RoundedRectangle (145,10 50x25), "ON", invisible if: m_Input_ROT.PS.STATE_OFF
    RoundedRectangle (145,10 50x25), "OFF", invisible if: m_Input_ROT.PS.STATE_ON
    Rectangle (5,50 100x30), "%s", text list: 'TextList_Moteurs', text index: 15
    Rectangle (10,3 125x25), "%s", text variable: m_Input_ROT.PS.Mnemo, text index: 15
    RoundedRectangle (105,50 100x30), "%1.0f rpm", text variable: m_Input_ROT.PRM_Vitesse, input disabled if: NOT MACHINE.STATE_Manu
        OnMouseDown: write the text variable via InputWithLimits, min m_Input_ROT.CONF_VMIN, max m_Input_ROT.CONF_VMAX, title 'Speed'
    RoundedRectangle (105,80 100x30), "%1.0f rpm", text variable: m_Input_ROT.PS.STATE_VIT
    Image (63,1 50x50), invisible if: NOT m_Input_ROT.STATE_NOK and Not m_Input_ROT.PS.STATE_NOK, image: MesImages.warning
    RoundedRectangle (140,5 60x35), invisible if: NOT MACHINE.STATE_Manu
        tap m_Input_ROT.M_On
    Rectangle (5,80 100x30), "%s", text list: 'TextList_Moteurs', text index: 7
END_VISUALIZATION

// ---- Visualizations/Symbole/MOUVEMENTS PS/VISU_VERIN_VH.TcVIS
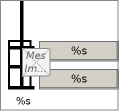
VISUALIZATION VISU_VERIN_VH  // 119x111
VAR_IN_OUT
	m_Input_VERIN: BLOCK_ACTUATOR;
	m_Input_MAINT: BOOL;
END_VAR
    Rectangle (8,40 23x49)
    Group (9,1 23x46), invisible if: NOT m_Input_VERIN.STATE_On
        Rectangle (0,45 25x3)
        Rectangle (11,0 3x47)
    Group (9,20 23x46), invisible if: (m_Input_VERIN.STATE_ON OR m_Input_VERIN.STATE_OFF) <> 0
        Rectangle (0,45 25x3)
        Rectangle (11,0 3x47)
    Group (9,41 23x46), invisible if: NOT m_Input_VERIN.STATE_OFF
        Rectangle (0,45 25x3)
        Rectangle (11,0 3x47)
    Rectangle (1,91 45x20), "%s", text variable: m_Input_VERIN.MNEMO
    Button (39,41 80x20), "%s", invisible if: NOT m_Input_VERIN.AUTOR_On_IHM OR NOT m_Input_MAINT, input disabled if: NOT m_Input_VERIN.AUTOR_On_IHM OR NOT m_Input_MAINT, text list: 'TextList_Orders', text index: 3
        tap m_Input_VERIN.M_On
    Button (39,69 80x20), "%s", invisible if: NOT m_Input_VERIN.AUTOR_Off_IHM OR NOT m_Input_MAINT, input disabled if: NOT m_Input_VERIN.AUTOR_Off_IHM OR NOT m_Input_MAINT, text list: 'TextList_Orders', text index: 2
        tap m_Input_VERIN.M_Off
    Image (22,48 28x28), invisible if: NOT m_Input_VERIN.STATE_NOK, image: MesImages.warning
END_VISUALIZATION

// ---- Visualizations/Symbole/POMPAGE/VISU_CONFIG_POMPAGE_CHAMBRE.TcVIS
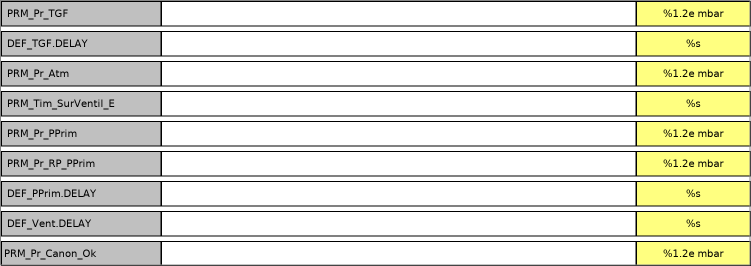
VISUALIZATION VISU_CONFIG_POMPAGE_CHAMBRE  // 751x266
VAR_IN_OUT
	m_Input_PRG_POMPAGE : BLOCK_PRG_POMPAGE;
END_VAR
    Rectangle (161,1 475x25), text list: 'TextList_Config_Pompage', text index: 2
    Rectangle (636,1 115x25), "%1.2e mbar", text variable: m_Input_PRG_POMPAGE.POMPAGE.PRM_Pr_TGF, input disabled if: NOT Global_Variables.PRG_USER.ACTU_USER.CONF_MACHINE
        OnMouseClick: write the text variable via InputWithLimits, min 10, max 1000
    Rectangle (1,1 160x25), "PRM_Pr_TGF"
    Rectangle (161,31 475x25), text list: 'TextList_Config_Pompage', text index: 3
    Rectangle (636,31 115x25), "%s", text variable: m_Input_PRG_POMPAGE.POMPAGE.DEF_TGF.DELAY, input disabled if: NOT Global_Variables.PRG_USER.ACTU_USER.CONF_MACHINE
        OnMouseClick: write the text variable via InputWithLimits
    Rectangle (1,31 160x25), "DEF_TGF.DELAY"
    Rectangle (161,61 475x25), text list: 'TextList_Config_Pompage', text index: 4
    Rectangle (161,91 475x25), text list: 'TextList_Config_Pompage', text index: 5
    Rectangle (636,61 115x25), "%1.2e mbar", text variable: m_Input_PRG_POMPAGE.POMPAGE.PRM_Pr_Atm, input disabled if: NOT Global_Variables.PRG_USER.ACTU_USER.CONF_MACHINE
        OnMouseClick: write the text variable via InputWithLimits, min 100, max 1000
    Rectangle (1,61 160x25), "PRM_Pr_Atm"
    Rectangle (636,91 115x25), "%s", text variable: m_Input_PRG_POMPAGE.POMPAGE.PRM_Tim_SurVentil_E, input disabled if: NOT Global_Variables.PRG_USER.ACTU_USER.CONF_MACHINE
        OnMouseClick: write the text variable via InputWithLimits
    Rectangle (1,91 160x25), "PRM_Tim_SurVentil_E"
    Rectangle (161,121 475x25), text list: 'TextList_Config_Pompage', text index: 6
    Rectangle (636,121 115x25), "%1.2e mbar", text variable: m_Input_PRG_POMPAGE.POMPAGE.PRM_Pr_PPrim, input disabled if: NOT Global_Variables.PRG_USER.ACTU_USER.CONF_MACHINE
        OnMouseClick: write the text variable via InputWithLimits, min 1e-3, max 2e-1
    Rectangle (1,121 160x25), "PRM_Pr_PPrim"
    Rectangle (1,151 160x25), "PRM_Pr_RP_PPrim"
    Rectangle (161,151 475x25), text list: 'TextList_Config_Pompage', text index: 7
    Rectangle (636,151 115x25), "%1.2e mbar", text variable: m_Input_PRG_POMPAGE.POMPAGE.PRM_Pr_RP_PPrim, input disabled if: NOT Global_Variables.PRG_USER.ACTU_USER.CONF_MACHINE
        OnMouseClick: write the text variable via InputWithLimits, min 1e-3, max 3e-1
    Rectangle (1,181 160x25), "DEF_PPrim.DELAY"
    Rectangle (161,181 475x25), text list: 'TextList_Config_Pompage', text index: 8
    Rectangle (636,181 115x25), "%s", text variable: m_Input_PRG_POMPAGE.POMPAGE.DEF_PPRIM.DELAY, input disabled if: NOT Global_Variables.PRG_USER.ACTU_USER.CONF_MACHINE
        OnMouseClick: write the text variable via InputWithLimits
    Rectangle (1,211 160x25), "DEF_Vent.DELAY"
    Rectangle (161,211 475x25), text list: 'TextList_Config_Pompage', text index: 9
    Rectangle (636,211 115x25), "%s", text variable: m_Input_PRG_POMPAGE.POMPAGE.DEF_VENT.DELAY, input disabled if: NOT Global_Variables.PRG_USER.ACTU_USER.CONF_MACHINE
        OnMouseClick: write the text variable via InputWithLimits
    Rectangle (1,241 160x25), "PRM_Pr_Canon_Ok"
    Rectangle (161,241 475x25), text list: 'TextList_Config_Pompage', text index: 10
    Rectangle (636,241 115x25), "%1.2e mbar", text variable: m_Input_PRG_POMPAGE.PRM_Pr_Canon_OK, input disabled if: NOT Global_Variables.PRG_USER.ACTU_USER.CONF_MACHINE
        OnMouseClick: write the text variable via InputWithLimits, min 0.000001, max 0.05
END_VISUALIZATION

// ---- Visualizations/Symbole/POMPAGE/VISU_CONFIG_POMPAGE_SAS.TcVIS
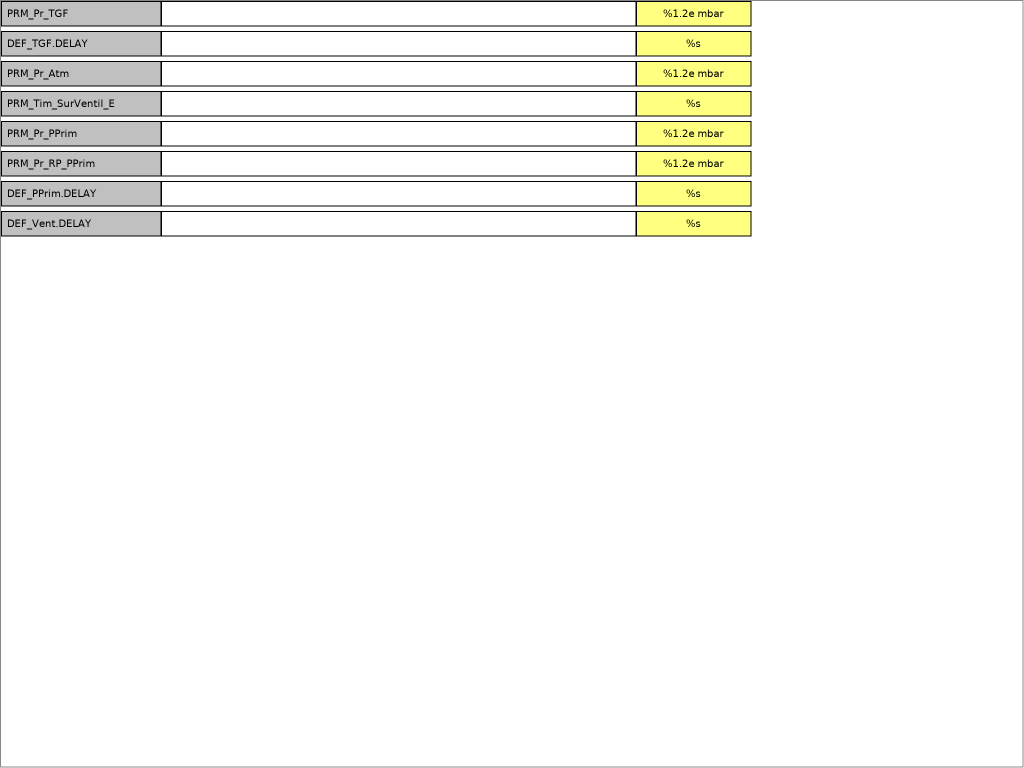
VISUALIZATION VISU_CONFIG_POMPAGE_SAS  // 1024x768
VAR_IN_OUT
	m_Input_PRG_POMPAGE : BLOCK_PRG_POMPAGE_SAS;
END_VAR
    Rectangle (161,1 475x25), text list: 'TextList_Config_Pompage', text index: 2
    Rectangle (636,1 115x25), "%1.2e mbar", text variable: m_Input_PRG_POMPAGE.POMPAGE.PRM_Pr_TGF, input disabled if: NOT Global_Variables.PRG_USER.ACTU_USER.CONF_MACHINE
        OnMouseClick: write the text variable via VisuDialogs.NumpadExtended, min 10, max 1000
    Rectangle (1,1 160x25), "PRM_Pr_TGF"
    Rectangle (161,31 475x25), text list: 'TextList_Config_Pompage', text index: 3
    Rectangle (636,31 115x25), "%s", text variable: m_Input_PRG_POMPAGE.POMPAGE.DEF_TGF.DELAY, input disabled if: NOT Global_Variables.PRG_USER.ACTU_USER.CONF_MACHINE
        OnMouseClick: write the text variable via VisuDialogs.Keypad
    Rectangle (1,31 160x25), "DEF_TGF.DELAY"
    Rectangle (161,61 475x25), text list: 'TextList_Config_Pompage', text index: 4
    Rectangle (161,91 475x25), text list: 'TextList_Config_Pompage', text index: 5
    Rectangle (636,61 115x25), "%1.2e mbar", text variable: m_Input_PRG_POMPAGE.POMPAGE.PRM_Pr_Atm, input disabled if: NOT Global_Variables.PRG_USER.ACTU_USER.CONF_MACHINE
        OnMouseClick: write the text variable via VisuDialogs.Numpad, min 100, max 1000
    Rectangle (1,61 160x25), "PRM_Pr_Atm"
    Rectangle (636,91 115x25), "%s", text variable: m_Input_PRG_POMPAGE.POMPAGE.PRM_Tim_SurVentil_E, input disabled if: NOT Global_Variables.PRG_USER.ACTU_USER.CONF_MACHINE
        OnMouseClick: write the text variable via VisuDialogs.Keypad
    Rectangle (1,91 160x25), "PRM_Tim_SurVentil_E"
    Rectangle (161,121 475x25), text list: 'TextList_Config_Pompage', text index: 6
    Rectangle (636,121 115x25), "%1.2e mbar", text variable: m_Input_PRG_POMPAGE.POMPAGE.PRM_Pr_PPrim, input disabled if: NOT Global_Variables.PRG_USER.ACTU_USER.CONF_MACHINE
        OnMouseClick: write the text variable via VisuDialogs.NumpadExtended, min 1e-3, max 1e-1
    Rectangle (1,121 160x25), "PRM_Pr_PPrim"
    Rectangle (1,151 160x25), "PRM_Pr_RP_PPrim"
    Rectangle (161,151 475x25), text list: 'TextList_Config_Pompage', text index: 7
    Rectangle (636,151 115x25), "%1.2e mbar", text variable: m_Input_PRG_POMPAGE.POMPAGE.PRM_Pr_RP_PPrim, input disabled if: NOT Global_Variables.PRG_USER.ACTU_USER.CONF_MACHINE
        OnMouseClick: write the text variable via VisuDialogs.NumpadExtended, min 1e-3, max 1e-1
    Rectangle (1,181 160x25), "DEF_PPrim.DELAY"
    Rectangle (161,181 475x25), text list: 'TextList_Config_Pompage', text index: 8
    Rectangle (636,181 115x25), "%s", text variable: m_Input_PRG_POMPAGE.POMPAGE.DEF_PPRIM.DELAY, input disabled if: NOT Global_Variables.PRG_USER.ACTU_USER.CONF_MACHINE
        OnMouseClick: write the text variable via VisuDialogs.Keypad
    Rectangle (1,211 160x25), "DEF_Vent.DELAY"
    Rectangle (161,211 475x25), text list: 'TextList_Config_Pompage', text index: 9
    Rectangle (636,211 115x25), "%s", text variable: m_Input_PRG_POMPAGE.POMPAGE.DEF_VENT.DELAY, input disabled if: NOT Global_Variables.PRG_USER.ACTU_USER.CONF_MACHINE
        OnMouseClick: write the text variable via VisuDialogs.Keypad
END_VISUALIZATION

// ---- Visualizations/Symbole/POMPAGE/VISU_CONFIG_VANNE_ASS_VVAT650.TcVIS
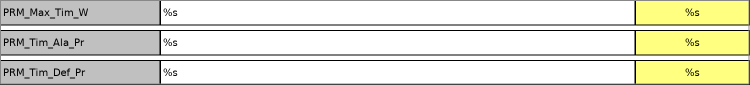
VISUALIZATION VISU_CONFIG_VANNE_ASS_VVAT650  // 750x85
(*visualistion pour secondaire dans chambre et primaire dans sas ==> paramètres pour chambre*)
VAR_IN_OUT
	m_Input_Vanne : BLOCK_VVAT_650_NO;
END_VAR
    Rectangle (160,0 475x25), "%s", text list: 'TextList_VVAT_650_ETHERCAT', text index: 1
    Rectangle (635,0 115x25), "%s", text variable: m_Input_Vanne.PRM_Max_Tim_W, input disabled if: NOT Global_Variables.PRG_USER.ACTU_USER.CONF_MACHINE
        OnMouseClick: write the text variable via Edit
    Rectangle (0,0 160x25), "PRM_Max_Tim_W"
    Rectangle (160,30 475x25), "%s", text list: 'TextList_VVAT_650_ETHERCAT', text index: 2
    Rectangle (635,30 115x25), "%s", text variable: m_Input_Vanne.PRM_Tim_Ala_Pr, input disabled if: NOT Global_Variables.PRG_USER.ACTU_USER.CONF_MACHINE
        OnMouseClick: write the text variable via Edit
    Rectangle (0,30 160x25), "PRM_Tim_Ala_Pr"
    Rectangle (0,60 160x25), "PRM_Tim_Def_Pr"
    Rectangle (160,60 475x25), "%s", text list: 'TextList_VVAT_650_ETHERCAT', text index: 3
    Rectangle (635,60 115x25), "%s", text variable: m_Input_Vanne.PRM_Tim_Def_Pr, input disabled if: NOT Global_Variables.PRG_USER.ACTU_USER.CONF_MACHINE
        OnMouseClick: write the text variable via Edit
END_VISUALIZATION

// ---- Visualizations/Symbole/POMPAGE/VISU_CONFIG_VANNE_ASS_VVAT653_ETHERCAT.TcVIS
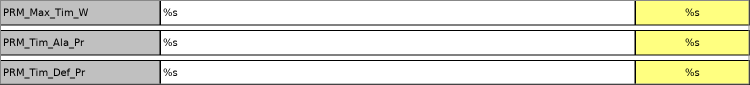
VISUALIZATION VISU_CONFIG_VANNE_ASS_VVAT653_ETHERCAT  // 750x85
(*visualistion pour secondaire dans chambre et primaire dans sas ==> paramètres pour chambre*)
VAR_IN_OUT
	m_Input_Vanne : BLOCK_VVAT_653_ETHERCAT;
END_VAR
    Rectangle (160,0 475x25), "%s", text list: 'TextList_VVAT_650_ETHERCAT', text index: 1
    Rectangle (635,0 115x25), "%s", text variable: m_Input_Vanne.PRM_Max_Tim_W, input disabled if: NOT Global_Variables.PRG_USER.ACTU_USER.CONF_MACHINE
        OnMouseClick: write the text variable via InputWithLimits
    Rectangle (0,0 160x25), "PRM_Max_Tim_W"
    Rectangle (160,30 475x25), "%s", text list: 'TextList_VVAT_650_ETHERCAT', text index: 2
    Rectangle (635,30 115x25), "%s", text variable: m_Input_Vanne.PRM_Tim_Ala_Pr, input disabled if: NOT Global_Variables.PRG_USER.ACTU_USER.CONF_MACHINE
        OnMouseClick: write the text variable via InputWithLimits
    Rectangle (0,30 160x25), "PRM_Tim_Ala_Pr"
    Rectangle (0,60 160x25), "PRM_Tim_Def_Pr"
    Rectangle (160,60 475x25), "%s", text list: 'TextList_VVAT_650_ETHERCAT', text index: 3
    Rectangle (635,60 115x25), "%s", text variable: m_Input_Vanne.PRM_Tim_Def_Pr, input disabled if: NOT Global_Variables.PRG_USER.ACTU_USER.CONF_MACHINE
        OnMouseClick: write the text variable via InputWithLimits
END_VISUALIZATION

// ---- Visualizations/Symbole/POMPAGE/VISU_CONFIG_INTERJOINT.TcVIS
